C07315=1211.113,371.634,-76.951,-175.920,7.915,148.347
C07316=1211.109,371.881,-76.984,-175.919,7.917,148.348
C07317=1211.105,372.129,-77.018,-175.918,7.920,148.348
C07318=1211.101,372.377,-77.052,-175.917,7.923,148.349
C07319=1211.097,372.625,-77.085,-175.915,7.926,148.349
C07320=1211.093,372.872,-77.119,-175.914,7.929,148.349
C07321=1211.089,373.120,-77.152,-175.912,7.932,148.350
C07322=1211.085,373.368,-77.185,-175.911,7.935,148.350
C07323=1211.080,373.615,-77.220,-175.910,7.938,148.351
C07324=1211.077,373.863,-77.253,-175.909,7.941,148.351
C07325=1211.073,374.111,-77.287,-175.908,7.944,148.351
C07326=1211.068,374.359,-77.321,-175.906,7.946,148.352
C07327=1211.064,374.606,-77.355,-175.905,7.949,148.352
C07328=1211.060,374.853,-77.388,-175.904,7.952,148.353
C07329=1211.057,375.102,-77.421,-175.903,7.956,148.353
C07330=1211.052,375.349,-77.456,-175.902,7.959,148.354
C07331=1211.048,375.597,-77.489,-175.900,7.962,148.354
C07332=1211.044,375.844,-77.523,-175.899,7.964,148.354
C07333=1211.040,376.093,-77.557,-175.898,7.967,148.355
C07334=1211.036,376.340,-77.591,-175.897,7.970,148.355
C07335=1211.032,376.588,-77.624,-175.896,7.973,148.356
C07336=1211.027,376.835,-77.658,-175.894,7.976,148.356
C07337=1211.023,377.083,-77.691,-175.893,7.978,148.356
C07338=1211.020,377.331,-77.726,-175.892,7.982,148.357
C07339=1211.015,377.578,-77.760,-175.891,7.984,148.357
C07340=1211.011,377.826,-77.793,-175.890,7.987,148.358
C07341=1211.007,378.073,-77.827,-175.889,7.990,148.358
C07342=1211.003,378.322,-77.861,-175.888,7.993,148.358
C07343=1210.999,378.569,-77.895,-175.886,7.996,148.359
C07344=1210.995,378.816,-77.928,-175.886,7.999,148.359
C07345=1210.991,379.065,-77.963,-175.885,8.002,148.360
C07346=1210.987,379.312,-77.997,-175.883,8.004,148.360
C07347=1210.982,379.560,-78.031,-175.882,8.007,148.361
C07348=1210.979,379.807,-78.065,-175.881,8.010,148.361
C07349=1210.975,380.055,-78.099,-175.880,8.013,148.362
C07350=1210.971,380.303,-78.133,-175.879,8.016,148.362
C07351=1210.967,380.550,-78.167,-175.878,8.019,148.362
C07352=1210.962,380.797,-78.201,-175.877,8.022,148.363
C07353=1210.959,381.046,-78.235,-175.876,8.025,148.363
C07354=1210.955,381.293,-78.268,-175.875,8.027,148.364
C07355=1210.950,381.540,-78.303,-175.874,8.029,148.364
C07356=1210.947,381.789,-78.336,-175.873,8.033,148.365
C07357=1210.942,382.036,-78.371,-175.872,8.035,148.365
C07358=1210.938,382.283,-78.405,-175.871,8.038,148.365
C07359=1210.933,382.531,-78.438,-175.870,8.041,148.366
C07360=1210.930,382.779,-78.473,-175.869,8.044,148.366
C07361=1210.926,383.026,-78.507,-175.868,8.047,148.367
C07362=1210.922,383.274,-78.541,-175.867,8.049,148.367
C07363=1210.917,383.522,-78.575,-175.866,8.052,148.368
C07364=1210.914,383.769,-78.609,-175.866,8.055,148.368
C07365=1210.909,384.017,-78.644,-175.864,8.058,148.369
C07366=1210.906,384.265,-78.678,-175.863,8.061,148.369
C07367=1210.901,384.513,-78.711,-175.862,8.064,148.370
C07368=1210.897,384.760,-78.745,-175.862,8.066,148.370
C07369=1210.893,385.008,-78.780,-175.861,8.069,148.371
C07370=1210.889,385.255,-78.814,-175.860,8.072,148.371
C07371=1210.885,385.502,-78.849,-175.859,8.075,148.372
C07372=1210.881,385.751,-78.882,-175.858,8.078,148.372
C07373=1210.877,385.998,-78.917,-175.857,8.080,148.372
C07374=1210.873,386.245,-78.950,-175.856,8.083,148.373
C07375=1210.869,386.493,-78.985,-175.855,8.086,148.373
C07376=1210.865,386.741,-79.019,-175.854,8.089,148.374
C07377=1210.860,386.988,-79.054,-175.854,8.091,148.374
C07378=1210.857,387.236,-79.088,-175.853,8.093,148.375
C07379=1210.852,387.484,-79.122,-175.852,8.097,148.375
C07380=1210.849,387.732,-79.156,-175.851,8.099,148.376
C07381=1210.845,387.979,-79.190,-175.850,8.102,148.376
C07382=1210.840,388.227,-79.225,-175.849,8.104,148.377
C07383=1210.837,388.474,-79.259,-175.848,8.108,148.377
C07384=1210.832,388.722,-79.293,-175.848,8.110,148.378
C07385=1210.828,388.969,-79.327,-175.847,8.113,148.378
C07386=1210.824,389.217,-79.362,-175.846,8.115,148.379
C07387=1210.821,389.464,-79.396,-175.846,8.118,148.379
C07388=1210.817,389.712,-79.431,-175.844,8.121,148.380
C07389=1210.812,389.960,-79.465,-175.844,8.124,148.380
C07390=1210.808,390.207,-79.499,-175.843,8.126,148.381
C07391=1210.804,390.455,-79.534,-175.842,8.129,148.381
C07392=1210.800,390.702,-79.568,-175.842,8.131,148.382
C07393=1210.796,390.950,-79.603,-175.841,8.134,148.382
C07394=1210.792,391.197,-79.637,-175.840,8.137,148.383
C07395=1210.788,391.445,-79.671,-175.839,8.139,148.383
C07396=1210.784,391.693,-79.706,-175.839,8.142,148.384
C07397=1210.779,391.940,-79.740,-175.838,8.144,148.384
C07398=1210.776,392.188,-79.775,-175.837,8.147,148.384
C07399=1210.771,392.470,-79.813,-175.837,8.150,148.385
C07400=1210.767,392.753,-79.853,-175.836,8.153,148.386
C07401=1210.762,393.035,-79.892,-175.835,8.156,148.386
C07402=1210.757,393.317,-79.932,-175.834,8.158,148.387
C07403=1210.753,393.564,-79.966,-175.834,8.161,148.387
C07404=1210.749,393.812,-80.000,-175.832,8.164,148.388
C07405=1210.745,394.060,-80.035,-175.832,8.167,148.388
C07406=1210.742,394.308,-80.069,-175.831,8.170,148.389
C07407=1210.737,394.555,-80.104,-175.831,8.172,148.389
C07408=1210.733,394.803,-80.138,-175.830,8.175,148.390
C07409=1210.729,395.050,-80.172,-175.829,8.177,148.390
C07410=1210.725,395.298,-80.207,-175.829,8.179,148.391
C07411=1210.721,395.546,-80.242,-175.828,8.182,148.391
C07412=1210.717,395.793,-80.277,-175.828,8.184,148.391
C07413=1210.713,396.040,-80.311,-175.827,8.187,148.392
C07414=1210.709,396.288,-80.345,-175.826,8.189,148.392
C07415=1210.705,396.536,-80.380,-175.826,8.192,148.393
C07416=1210.701,396.783,-80.414,-175.825,8.195,148.394
C07417=1210.697,397.031,-80.449,-175.824,8.197,148.394
C07418=1210.692,397.279,-80.483,-175.824,8.200,148.394
C07419=1210.688,397.525,-80.519,-175.824,8.202,148.395
C07420=1210.685,397.773,-80.553,-175.823,8.205,148.395
C07421=1210.680,398.021,-80.587,-175.822,8.207,148.396
C07422=1210.676,398.269,-80.622,-175.822,8.210,148.397
C07423=1210.672,398.516,-80.657,-175.821,8.212,148.397
C07424=1210.669,398.764,-80.691,-175.821,8.214,148.397
C07425=1210.664,399.011,-80.726,-175.820,8.217,148.398
C07426=1210.660,399.259,-80.761,-175.819,8.219,148.398
C07427=1210.656,399.506,-80.795,-175.819,8.222,148.399
C07428=1210.653,399.754,-80.830,-175.818,8.224,148.399
C07429=1210.648,400.001,-80.865,-175.818,8.227,148.400
C07430=1210.644,400.249,-80.900,-175.818,8.229,148.400
C07431=1210.640,400.496,-80.934,-175.816,8.232,148.401
C07432=1210.636,400.744,-80.968,-175.816,8.234,148.401
C07433=1210.632,400.992,-81.003,-175.816,8.236,148.402
C07434=1210.628,401.239,-81.038,-175.815,8.239,148.402
C07435=1210.624,401.487,-81.073,-175.815,8.241,148.403
C07436=1210.620,401.735,-81.108,-175.814,8.244,148.403
C07437=1210.616,401.981,-81.142,-175.814,8.246,148.404
C07438=1210.612,402.229,-81.177,-175.813,8.249,148.404
C07439=1210.608,402.477,-81.212,-175.813,8.251,148.405
C07440=1210.604,402.725,-81.246,-175.812,8.253,148.405
C07441=1210.599,402.972,-81.282,-175.812,8.255,148.406
C07442=1210.595,403.220,-81.316,-175.811,8.258,148.406
C07443=1210.592,403.467,-81.350,-175.810,8.260,148.407
C07444=1210.588,403.714,-81.386,-175.810,8.263,148.407
C07445=1210.583,403.962,-81.420,-175.810,8.265,148.408
C07446=1210.579,404.210,-81.455,-175.809,8.268,148.408
C07447=1210.575,404.457,-81.490,-175.809,8.270,148.409
C07448=1210.571,404.705,-81.525,-175.808,8.272,148.409
C07449=1210.568,404.953,-81.559,-175.808,8.274,148.409
C07450=1210.564,405.200,-81.595,-175.807,8.277,148.410
C07451=1210.560,405.448,-81.629,-175.807,8.280,148.411
C07452=1210.555,405.695,-81.664,-175.806,8.282,148.411
C07453=1210.551,405.943,-81.699,-175.806,8.284,148.411
C07454=1210.547,406.190,-81.734,-175.806,8.286,148.412
C07455=1210.544,406.438,-81.768,-175.805,8.288,148.412
C07456=1210.539,406.685,-81.803,-175.805,8.290,148.413
C07457=1210.535,406.933,-81.838,-175.804,8.293,148.413
C07458=1210.531,407.179,-81.873,-175.803,8.295,148.414
C07459=1210.527,407.428,-81.908,-175.803,8.298,148.414
C07460=1210.523,407.676,-81.943,-175.803,8.300,148.415
C07461=1210.519,407.923,-81.978,-175.802,8.302,148.415
C07462=1210.515,408.171,-82.013,-175.802,8.304,148.416
C07463=1210.511,408.417,-82.048,-175.802,8.306,148.416
C07464=1210.508,408.665,-82.082,-175.801,8.309,148.417
C07465=1210.503,408.912,-82.118,-175.800,8.312,148.417
C07466=1210.499,409.160,-82.152,-175.800,8.314,148.417
C07467=1210.495,409.408,-82.187,-175.800,8.316,148.418
C07468=1210.491,409.655,-82.222,-175.799,8.318,148.419
C07469=1210.487,409.903,-82.257,-175.799,8.320,148.419
C07470=1210.483,410.150,-82.292,-175.798,8.322,148.419
C07471=1210.479,410.398,-82.327,-175.798,8.325,148.420
C07472=1210.475,410.645,-82.362,-175.798,8.327,148.420
C07473=1210.471,410.893,-82.397,-175.797,8.329,148.421
C07474=1210.467,411.141,-82.433,-175.797,8.331,148.421
C07475=1210.463,411.388,-82.467,-175.797,8.333,148.422
C07476=1210.459,411.635,-82.502,-175.796,8.335,148.422
C07477=1210.455,411.883,-82.537,-175.796,8.338,148.423
C07478=1210.451,412.130,-82.572,-175.795,8.340,148.423
C07479=1210.447,412.378,-82.607,-175.795,8.343,148.424
C07480=1210.443,412.625,-82.642,-175.794,8.345,148.424
C07481=1210.439,412.873,-82.677,-175.794,8.347,148.425
C07482=1210.435,413.120,-82.712,-175.794,8.349,148.425
C07483=1210.431,413.368,-82.747,-175.793,8.351,148.425
C07484=1210.427,413.616,-82.783,-175.793,8.353,148.426
C07485=1210.423,413.863,-82.817,-175.793,8.356,148.426
C07486=1210.419,414.110,-82.853,-175.792,8.358,148.427
C07487=1210.414,414.358,-82.887,-175.792,8.360,148.427
C07488=1210.411,414.605,-82.923,-175.791,8.362,148.428
C07489=1210.407,414.853,-82.958,-175.791,8.364,148.428
C07490=1210.402,415.100,-82.993,-175.791,8.366,148.429
C07491=1210.399,415.348,-83.028,-175.790,8.368,148.429
C07492=1210.394,415.595,-83.063,-175.790,8.371,148.430
C07493=1210.391,415.843,-83.098,-175.789,8.373,148.430
C07494=1210.387,416.091,-83.133,-175.789,8.375,148.430
C07495=1210.383,416.341,-83.169,-175.789,8.377,148.431
C07496=1210.379,416.592,-83.204,-175.788,8.379,148.431
C07497=1210.377,416.842,-83.239,-175.788,8.381,148.432
C07498=1210.379,417.093,-83.274,-175.788,8.383,148.432
C07499=1209.957,417.093,-83.312,-175.791,8.393,148.436
C07500=1209.956,416.839,-83.276,-175.791,8.392,148.436
C07501=1209.957,416.587,-83.240,-175.791,8.390,148.435
C07502=1209.961,416.333,-83.204,-175.791,8.388,148.435
C07503=1209.965,416.080,-83.168,-175.792,8.386,148.434
C07504=1209.969,415.832,-83.133,-175.792,8.383,148.434
C07505=1209.973,415.585,-83.098,-175.793,8.381,148.433
C07506=1209.977,415.337,-83.063,-175.793,8.379,148.433
C07507=1209.981,415.090,-83.028,-175.793,8.377,148.432
C07508=1209.985,414.842,-82.993,-175.794,8.375,148.432
C07509=1209.989,414.594,-82.957,-175.794,8.373,148.431
C07510=1209.993,414.347,-82.922,-175.794,8.370,148.431
C07511=1209.997,414.099,-82.887,-175.795,8.368,148.431
C07512=1210.001,413.853,-82.852,-175.795,8.366,148.430
C07513=1210.005,413.604,-82.817,-175.796,8.364,148.430
C07514=1210.009,413.357,-82.782,-175.796,8.362,148.429
C07515=1210.013,413.109,-82.747,-175.796,8.360,148.429
C07516=1210.017,412.862,-82.712,-175.797,8.358,148.428
C07517=1210.022,412.615,-82.677,-175.797,8.355,148.428
C07518=1210.025,412.367,-82.642,-175.798,8.353,148.427
C07519=1210.029,412.119,-82.607,-175.798,8.351,148.427
C07520=1210.034,411.872,-82.572,-175.798,8.349,148.426
C07521=1210.038,411.624,-82.537,-175.799,8.347,148.426
C07522=1210.042,411.377,-82.502,-175.800,8.344,148.425
C07523=1210.045,411.129,-82.467,-175.800,8.341,148.425
C07524=1210.049,410.882,-82.432,-175.801,8.339,148.425
C07525=1210.053,410.635,-82.397,-175.801,8.337,148.424
C07526=1210.057,410.387,-82.362,-175.801,8.335,148.423
C07527=1210.061,410.140,-82.327,-175.802,8.333,148.423
C07528=1210.065,409.892,-82.292,-175.802,8.331,148.423
C07529=1210.070,409.645,-82.257,-175.802,8.328,148.422
C07530=1210.073,409.397,-82.222,-175.803,8.326,148.422
C07531=1210.077,409.149,-82.187,-175.803,8.324,148.421
C07532=1210.082,408.902,-82.152,-175.803,8.322,148.421
C07533=1210.086,408.654,-82.117,-175.804,8.320,148.420
C07534=1210.090,408.407,-82.082,-175.804,8.318,148.420
C07535=1210.093,408.160,-82.048,-175.805,8.315,148.419
C07536=1210.098,407.912,-82.013,-175.806,8.313,148.419
C07537=1210.101,407.665,-81.978,-175.806,8.310,148.418
C07538=1210.105,407.416,-81.943,-175.806,8.308,148.418
C07539=1210.110,407.170,-81.908,-175.807,8.306,148.417
C07540=1210.114,406.922,-81.873,-175.807,8.304,148.417
C07541=1210.118,406.675,-81.838,-175.807,8.302,148.416
C07542=1210.122,406.427,-81.803,-175.808,8.299,148.416
C07543=1210.126,406.180,-81.769,-175.809,8.296,148.415
C07544=1210.129,405.932,-81.733,-175.809,8.294,148.415
C07545=1210.134,405.685,-81.699,-175.809,8.292,148.415
C07546=1210.138,405.436,-81.664,-175.810,8.290,148.414
C07547=1210.141,405.189,-81.628,-175.810,8.288,148.414
C07548=1210.146,404.942,-81.594,-175.811,8.285,148.413
C07549=1210.150,404.694,-81.558,-175.811,8.283,148.413
C07550=1210.154,404.447,-81.525,-175.811,8.280,148.412
C07551=1210.157,404.199,-81.490,-175.812,8.278,148.412
C07552=1210.162,403.952,-81.455,-175.812,8.276,148.411
C07553=1210.166,403.704,-81.420,-175.813,8.273,148.411
C07554=1210.170,403.456,-81.385,-175.814,8.271,148.410
C07555=1210.174,403.209,-81.350,-175.814,8.269,148.410
C07556=1210.178,402.962,-81.316,-175.814,8.266,148.409
C07557=1210.182,402.714,-81.281,-175.815,8.264,148.409
C07558=1210.186,402.466,-81.247,-175.816,8.261,148.408
C07559=1210.190,402.219,-81.211,-175.816,8.259,148.408
C07560=1210.195,401.971,-81.177,-175.816,8.257,148.407
C07561=1210.199,401.723,-81.142,-175.817,8.254,148.407
C07562=1210.202,401.477,-81.107,-175.817,8.252,148.406
C07563=1210.206,401.229,-81.072,-175.818,8.250,148.406
C07564=1210.211,400.981,-81.038,-175.819,8.247,148.405
C07565=1210.215,400.733,-81.003,-175.819,8.244,148.405
C07566=1210.219,400.486,-80.968,-175.820,8.242,148.404
C07567=1210.222,400.239,-80.934,-175.820,8.240,148.404
C07568=1210.227,399.991,-80.899,-175.821,8.237,148.403
C07569=1210.231,399.743,-80.864,-175.821,8.235,148.403
C07570=1210.235,399.496,-80.829,-175.822,8.233,148.402
C07571=1210.238,399.248,-80.795,-175.822,8.230,148.402
C07572=1210.243,399.001,-80.760,-175.823,8.228,148.402
C07573=1210.247,398.753,-80.726,-175.824,8.225,148.401
C07574=1210.251,398.505,-80.691,-175.824,8.222,148.400
C07575=1210.254,398.258,-80.656,-175.825,8.220,148.400
C07576=1210.259,398.011,-80.622,-175.825,8.217,148.399
C07577=1210.263,397.763,-80.587,-175.826,8.215,148.399
C07578=1210.267,397.515,-80.552,-175.826,8.213,148.399
C07579=1210.270,397.267,-80.518,-175.827,8.210,148.398
C07580=1210.275,397.021,-80.483,-175.827,8.208,148.397
C07581=1210.279,396.773,-80.448,-175.828,8.205,148.397
C07582=1210.283,396.525,-80.414,-175.829,8.203,148.397
C07583=1210.286,396.277,-80.379,-175.829,8.199,148.396
C07584=1210.291,396.030,-80.345,-175.830,8.198,148.396
C07585=1210.295,395.782,-80.310,-175.830,8.195,148.395
C07586=1210.300,395.534,-80.276,-175.831,8.192,148.395
C07587=1210.303,395.287,-80.242,-175.832,8.190,148.394
C07588=1210.307,395.040,-80.206,-175.832,8.187,148.394
C07589=1210.312,394.792,-80.172,-175.833,8.185,148.393
C07590=1210.315,394.545,-80.138,-175.834,8.182,148.393
C07591=1210.319,394.297,-80.103,-175.834,8.180,148.392
C07592=1210.323,394.049,-80.068,-175.835,8.177,148.392
C07593=1210.327,393.802,-80.034,-175.835,8.175,148.391
C07594=1210.331,393.554,-80.000,-175.837,8.172,148.391
C07595=1210.336,393.306,-79.965,-175.837,8.170,148.390
C07596=1210.340,393.024,-79.925,-175.838,8.166,148.390
C07597=1210.345,392.742,-79.887,-175.838,8.163,148.389
C07598=1210.349,392.460,-79.847,-175.839,8.161,148.389
C07599=1210.354,392.177,-79.809,-175.840,8.157,148.388
C07600=1210.358,391.929,-79.774,-175.840,8.155,148.387
C07601=1210.363,391.682,-79.739,-175.842,8.152,148.387
C07602=1210.366,391.434,-79.705,-175.842,8.149,148.386
C07603=1210.370,391.187,-79.671,-175.843,8.147,148.386
C07604=1210.374,390.940,-79.637,-175.844,8.144,148.386
C07605=1210.378,390.691,-79.602,-175.844,8.142,148.385
C07606=1210.383,390.444,-79.567,-175.845,8.139,148.385
C07607=1210.386,390.196,-79.533,-175.846,8.136,148.384
C07608=1210.390,389.949,-79.499,-175.847,8.134,148.384
C07609=1210.395,389.701,-79.464,-175.847,8.131,148.383
C07610=1210.398,389.454,-79.430,-175.849,8.128,148.383
C07611=1210.403,389.206,-79.396,-175.849,8.126,148.382
C07612=1210.406,388.958,-79.361,-175.850,8.123,148.382
C07613=1210.411,388.711,-79.327,-175.851,8.120,148.381
C07614=1210.415,388.464,-79.293,-175.851,8.118,148.381
C07615=1210.418,388.216,-79.258,-175.852,8.115,148.380
C07616=1210.423,387.968,-79.224,-175.853,8.112,148.380
C07617=1210.427,387.721,-79.190,-175.854,8.110,148.379
C07618=1210.431,387.473,-79.155,-175.855,8.107,148.379
C07619=1210.435,387.226,-79.121,-175.856,8.104,148.378
C07620=1210.439,386.977,-79.087,-175.856,8.102,148.378
C07621=1210.443,386.730,-79.053,-175.857,8.099,148.377
C07622=1210.447,386.483,-79.019,-175.858,8.096,148.377
C07623=1210.451,386.235,-78.984,-175.859,8.093,148.376
C07624=1210.455,385.987,-78.950,-175.860,8.091,148.376
C07625=1210.460,385.740,-78.915,-175.860,8.088,148.375
C07626=1210.463,385.492,-78.881,-175.861,8.085,148.375
C07627=1210.468,385.244,-78.847,-175.862,8.082,148.374
C07628=1210.472,384.997,-78.814,-175.863,8.079,148.374
C07629=1210.476,384.749,-78.779,-175.864,8.077,148.374
C07630=1210.479,384.502,-78.745,-175.865,8.074,148.373
C07631=1210.484,384.254,-78.710,-175.866,8.071,148.373
C07632=1210.488,384.006,-78.677,-175.867,8.068,148.372
C07633=1210.492,383.759,-78.642,-175.868,8.065,148.372
C07634=1210.496,383.511,-78.609,-175.869,8.062,148.371
C07635=1210.500,383.263,-78.574,-175.869,8.060,148.371
C07636=1210.504,383.016,-78.540,-175.871,8.057,148.370
C07637=1210.509,382.768,-78.506,-175.872,8.054,148.370
C07638=1210.512,382.520,-78.472,-175.873,8.051,148.369
C07639=1210.516,382.273,-78.438,-175.874,8.049,148.369
C07640=1210.521,382.025,-78.404,-175.875,8.046,148.369
C07641=1210.524,381.777,-78.370,-175.876,8.043,148.368
C07642=1210.528,381.530,-78.336,-175.876,8.041,148.368
C07643=1210.532,381.283,-78.302,-175.878,8.038,148.367
C07644=1210.537,381.035,-78.268,-175.878,8.035,148.367
C07645=1210.540,380.787,-78.234,-175.880,8.032,148.366
C07646=1210.545,380.540,-78.199,-175.881,8.029,148.366
C07647=1210.549,380.292,-78.166,-175.881,8.026,148.365
C07648=1210.552,380.044,-78.132,-175.883,8.023,148.365
C07649=1210.557,379.797,-78.097,-175.884,8.020,148.365
C07650=1210.561,379.549,-78.064,-175.885,8.018,148.364
C07651=1210.566,379.301,-78.030,-175.886,8.014,148.364
C07652=1210.569,379.053,-77.996,-175.887,8.012,148.363
C07653=1210.573,378.806,-77.962,-175.888,8.009,148.363
C07654=1210.577,378.559,-77.928,-175.889,8.006,148.362
C07655=1210.582,378.311,-77.895,-175.891,8.003,148.362
C07656=1210.586,378.063,-77.860,-175.891,8.000,148.361
C07657=1210.590,377.815,-77.827,-175.893,7.997,148.361
C07658=1210.594,377.568,-77.793,-175.894,7.994,148.361
C07659=1210.598,377.320,-77.758,-175.895,7.992,148.360
C07660=1210.602,377.072,-77.725,-175.896,7.989,148.360
C07661=1210.605,376.825,-77.691,-175.897,7.986,148.359
C07662=1210.610,376.577,-77.657,-175.898,7.983,148.359
C07663=1210.614,376.330,-77.623,-175.899,7.980,148.358
C07664=1210.618,376.081,-77.590,-175.901,7.977,148.358
C07665=1210.622,375.834,-77.555,-175.902,7.974,148.358
C07666=1210.626,375.586,-77.522,-175.903,7.972,148.357
C07667=1210.630,375.339,-77.488,-175.904,7.969,148.357
C07668=1210.635,375.090,-77.454,-175.905,7.966,148.357
C07669=1210.638,374.843,-77.420,-175.907,7.962,148.356
C07670=1210.643,374.595,-77.387,-175.908,7.960,148.356
C07671=1210.646,374.348,-77.353,-175.909,7.957,148.355
C07672=1210.651,374.100,-77.320,-175.910,7.954,148.355
C07673=1210.654,373.853,-77.285,-175.911,7.951,148.354
C07674=1210.659,373.605,-77.252,-175.913,7.948,148.354
C07675=1210.663,373.357,-77.218,-175.914,7.945,148.354
C07676=1210.667,373.110,-77.185,-175.915,7.942,148.353
C07677=1210.671,372.862,-77.151,-175.917,7.939,148.353
C07678=1210.675,372.614,-77.117,-175.918,7.936,148.352
C07679=1210.679,372.366,-77.084,-175.919,7.933,148.352
C07680=1210.684,372.118,-77.050,-175.920,7.930,148.352
C07681=1210.688,371.871,-77.016,-175.922,7.928,148.351
C07682=1210.692,371.623,-76.983,-175.923,7.925,148.351
C07683=1210.696,371.376,-76.950,-175.925,7.921,148.350
C07684=1210.700,371.128,-76.915,-175.926,7.919,148.350
C07685=1210.704,370.880,-76.882,-175.927,7.916,148.350
C07686=1210.708,370.632,-76.849,-175.929,7.913,148.349
C07687=1210.712,370.385,-76.815,-175.930,7.910,148.349
C07688=1210.716,370.137,-76.782,-175.932,7.906,148.348
C07689=1210.721,369.889,-76.748,-175.933,7.904,148.348
C07690=1210.724,369.641,-76.714,-175.934,7.901,148.348
C07691=1210.728,369.394,-76.681,-175.936,7.898,148.348
C07692=1210.732,369.146,-76.648,-175.937,7.895,148.347
C07693=1210.737,368.898,-76.614,-175.939,7.892,148.347
C07694=1210.740,368.651,-76.581,-175.940,7.889,148.346
C07695=1210.745,368.403,-76.547,-175.941,7.886,148.346
C07696=1210.749,368.155,-76.514,-175.943,7.883,148.345
C07697=1210.754,367.908,-76.481,-175.944,7.880,148.345
C07698=1210.757,367.659,-76.447,-175.946,7.877,148.345
C07699=1210.761,367.412,-76.413,-175.947,7.874,148.344
C07700=1210.766,367.132,-76.376,-175.948,7.871,148.344
C07701=1210.771,366.851,-76.338,-175.950,7.867,148.344
C07702=1210.775,366.572,-76.300,-175.952,7.864,148.343
C07703=1210.779,366.291,-76.263,-175.954,7.861,148.343
C07704=1210.784,366.043,-76.229,-175.955,7.857,148.343
C07705=1210.788,365.796,-76.195,-175.957,7.855,148.342
C07706=1210.792,365.548,-76.162,-175.958,7.852,148.342
C07707=1210.796,365.300,-76.129,-175.960,7.848,148.341
C07708=1210.801,365.052,-76.096,-175.961,7.846,148.341
C07709=1210.805,364.805,-76.063,-175.963,7.843,148.341
C07710=1210.809,364.557,-76.030,-175.965,7.839,148.340
C07711=1210.813,364.309,-75.997,-175.966,7.837,148.340
C07712=1210.817,364.061,-75.963,-175.967,7.834,148.340
C07713=1210.821,363.813,-75.930,-175.969,7.830,148.339
C07714=1210.825,363.565,-75.897,-175.971,7.828,148.339
C07715=1210.829,363.318,-75.864,-175.972,7.825,148.339
C07716=1210.833,363.070,-75.830,-175.974,7.821,148.338
C07717=1210.837,362.822,-75.797,-175.975,7.819,148.338
C07718=1210.841,362.574,-75.764,-175.977,7.815,148.338
C07719=1210.845,362.327,-75.731,-175.979,7.813,148.338
C07720=1210.850,362.079,-75.698,-175.980,7.810,148.337
C07721=1210.854,361.831,-75.665,-175.982,7.807,148.337
C07722=1210.858,361.584,-75.631,-175.983,7.804,148.337
C07723=1210.862,361.336,-75.598,-175.985,7.801,148.336
C07724=1210.866,361.088,-75.565,-175.987,7.798,148.336
C07725=1210.870,360.840,-75.532,-175.988,7.795,148.336
C07726=1210.874,360.593,-75.499,-175.990,7.791,148.335
C07727=1210.878,360.345,-75.466,-175.992,7.789,148.335
C07728=1210.882,360.098,-75.433,-175.994,7.785,148.335
C07729=1210.886,359.850,-75.400,-175.995,7.783,148.335
C07730=1210.891,359.601,-75.368,-175.996,7.780,148.334
C07731=1210.895,359.354,-75.334,-175.999,7.777,148.334
C07732=1210.899,359.106,-75.301,-176.000,7.774,148.334
C07733=1210.903,358.858,-75.268,-176.002,7.770,148.333
C07734=1210.907,358.611,-75.235,-176.004,7.768,148.333
C07735=1210.911,358.363,-75.202,-176.005,7.764,148.333
C07736=1210.915,358.115,-75.170,-176.007,7.762,148.333
C07737=1210.919,357.867,-75.137,-176.008,7.759,148.332
C07738=1210.923,357.619,-75.104,-176.011,7.756,148.332
C07739=1210.927,357.372,-75.070,-176.012,7.753,148.332
C07740=1210.932,357.123,-75.038,-176.014,7.749,148.331
C07741=1210.936,356.875,-75.005,-176.016,7.747,148.331
C07742=1210.940,356.628,-74.972,-176.018,7.744,148.331
C07743=1210.943,356.380,-74.939,-176.019,7.741,148.330
C07744=1210.949,356.133,-74.907,-176.021,7.737,148.330
C07745=1210.953,355.885,-74.874,-176.023,7.735,148.330
C07746=1210.957,355.637,-74.841,-176.025,7.732,148.330
C07747=1210.961,355.389,-74.808,-176.026,7.729,148.329
C07748=1210.965,355.141,-74.776,-176.028,7.726,148.329
C07749=1210.969,354.894,-74.743,-176.030,7.723,148.329
C07750=1210.973,354.645,-74.710,-176.031,7.720,148.329
C07751=1210.977,354.398,-74.677,-176.034,7.717,148.328
C07752=1210.981,354.150,-74.644,-176.035,7.714,148.328
C07753=1210.985,353.902,-74.612,-176.037,7.711,148.328
C07754=1210.989,353.654,-74.579,-176.039,7.708,148.328
C07755=1210.994,353.407,-74.547,-176.041,7.705,148.327
C07756=1210.998,353.159,-74.514,-176.042,7.702,148.327
C07757=1211.002,352.911,-74.481,-176.045,7.699,148.327
C07758=1211.006,352.663,-74.449,-176.046,7.696,148.327
C07759=1211.011,352.415,-74.415,-176.048,7.693,148.327
C07760=1211.014,352.167,-74.384,-176.050,7.690,148.326
C07761=1211.018,351.920,-74.350,-176.052,7.687,148.326
C07762=1211.023,351.671,-74.318,-176.054,7.684,148.326
C07763=1211.027,351.424,-74.286,-176.056,7.681,148.326
C07764=1211.031,351.176,-74.253,-176.057,7.678,148.325
C07765=1211.035,350.928,-74.220,-176.060,7.675,148.325
C07766=1211.039,350.680,-74.188,-176.061,7.672,148.325
C07767=1211.043,350.433,-74.155,-176.063,7.669,148.325
C07768=1211.048,350.184,-74.123,-176.065,7.666,148.324
C07769=1211.052,349.938,-74.091,-176.067,7.663,148.324
C07770=1211.056,349.689,-74.058,-176.068,7.660,148.324
C07771=1211.061,349.441,-74.026,-176.071,7.657,148.324
C07772=1211.064,349.193,-73.993,-176.072,7.655,148.324
C07773=1211.068,348.945,-73.961,-176.075,7.651,148.323
C07774=1211.073,348.698,-73.928,-176.076,7.649,148.323
C07775=1211.077,348.450,-73.896,-176.078,7.645,148.323
C07776=1211.081,348.202,-73.864,-176.080,7.643,148.323
C07777=1211.085,347.954,-73.831,-176.082,7.640,148.322
C07778=1211.089,347.706,-73.799,-176.084,7.637,148.322
C07779=1211.093,347.459,-73.767,-176.086,7.634,148.322
C07780=1211.098,347.211,-73.734,-176.088,7.631,148.322
C07781=1211.102,346.962,-73.702,-176.090,7.628,148.322
C07782=1211.106,346.714,-73.670,-176.092,7.625,148.321
C07783=1211.110,346.466,-73.637,-176.094,7.622,148.321
C07784=1211.114,346.219,-73.605,-176.095,7.619,148.321
C07785=1211.119,345.971,-73.573,-176.098,7.616,148.321
C07786=1211.122,345.723,-73.541,-176.099,7.614,148.321
C07787=1211.127,345.475,-73.508,-176.102,7.610,148.320
C07788=1211.131,345.228,-73.476,-176.103,7.608,148.320
C07789=1211.135,344.980,-73.444,-176.105,7.604,148.320
C07790=1211.139,344.732,-73.412,-176.107,7.602,148.320
C07791=1211.144,344.484,-73.380,-176.109,7.599,148.320
C07792=1211.148,344.236,-73.348,-176.111,7.596,148.319
C07793=1211.152,343.988,-73.315,-176.113,7.593,148.319
C07794=1211.156,343.740,-73.283,-176.115,7.590,148.319
C07795=1211.161,343.492,-73.251,-176.117,7.587,148.319
C07796=1211.164,343.244,-73.219,-176.120,7.584,148.319
C07797=1211.169,342.996,-73.187,-176.121,7.581,148.319
C07798=1211.173,342.749,-73.155,-176.124,7.578,148.318
C07799=1211.177,342.500,-73.123,-176.125,7.575,148.318
C07800=1211.181,342.252,-73.091,-176.127,7.572,148.318
C07801=1211.185,342.004,-73.059,-176.129,7.570,148.318
C07802=1211.190,341.757,-73.026,-176.131,7.566,148.318
C07803=1211.193,341.509,-72.994,-176.133,7.564,148.318
C07804=1211.199,341.231,-72.959,-176.136,7.561,148.317
C07805=1211.203,340.953,-72.923,-176.138,7.557,148.317
C07806=1211.207,340.675,-72.887,-176.140,7.554,148.317
C07807=1211.213,340.396,-72.851,-176.142,7.551,148.317
C07808=1211.217,340.148,-72.819,-176.145,7.548,148.317
C07809=1211.221,339.901,-72.788,-176.146,7.545,148.317
C07810=1211.225,339.652,-72.755,-176.149,7.542,148.316
C07811=1211.229,339.404,-72.724,-176.150,7.539,148.316
C07812=1211.233,339.157,-72.692,-176.153,7.536,148.316
C07813=1211.238,338.909,-72.660,-176.155,7.534,148.316
C07814=1211.242,338.661,-72.628,-176.157,7.530,148.316
C07815=1211.246,338.413,-72.596,-176.159,7.528,148.316
C07816=1211.250,338.165,-72.564,-176.161,7.524,148.315
C07817=1211.255,337.918,-72.532,-176.163,7.522,148.315
C07818=1211.258,337.670,-72.501,-176.165,7.519,148.315
C07819=1211.262,337.422,-72.469,-176.167,7.515,148.315
C07820=1211.267,337.173,-72.437,-176.169,7.513,148.315
C07821=1211.271,336.925,-72.406,-176.172,7.510,148.315
C07822=1211.275,336.678,-72.374,-176.173,7.507,148.315
C07823=1211.279,336.430,-72.342,-176.175,7.504,148.314
C07824=1211.283,336.182,-72.310,-176.178,7.502,148.314
C07825=1211.288,335.934,-72.279,-176.180,7.498,148.314
C07826=1211.292,335.686,-72.247,-176.181,7.496,148.314
C07827=1211.296,335.438,-72.216,-176.184,7.493,148.314
C07828=1211.301,335.190,-72.183,-176.186,7.490,148.314
C07829=1211.305,334.943,-72.152,-176.188,7.487,148.314
C07830=1211.309,334.694,-72.121,-176.191,7.484,148.314
C07831=1211.313,334.446,-72.089,-176.192,7.481,148.313
C07832=1211.317,334.198,-72.057,-176.194,7.478,148.313
C07833=1211.321,333.950,-72.026,-176.197,7.476,148.313
C07834=1211.326,333.702,-71.994,-176.199,7.473,148.313
C07835=1211.330,333.454,-71.962,-176.201,7.470,148.313
C07836=1211.334,333.206,-71.931,-176.203,7.467,148.313
C07837=1211.338,332.958,-71.900,-176.205,7.465,148.313
C07838=1211.342,332.711,-71.868,-176.207,7.461,148.313
C07839=1211.346,332.462,-71.837,-176.210,7.458,148.312
C07840=1211.351,332.215,-71.806,-176.212,7.456,148.312
C07841=1211.355,331.966,-71.773,-176.214,7.453,148.312
C07842=1211.360,331.719,-71.742,-176.216,7.450,148.312
C07843=1211.363,331.470,-71.710,-176.218,7.447,148.312
C07844=1211.368,331.223,-71.680,-176.220,7.444,148.312
C07845=1211.372,330.974,-71.648,-176.223,7.441,148.312
C07846=1211.376,330.727,-71.617,-176.224,7.439,148.312
C07847=1211.380,330.478,-71.585,-176.227,7.436,148.312
C07848=1211.385,330.231,-71.555,-176.229,7.433,148.312
C07849=1211.388,329.982,-71.523,-176.231,7.430,148.312
C07850=1211.393,329.735,-71.492,-176.233,7.427,148.311
C07851=1211.397,329.486,-71.460,-176.236,7.425,148.311
C07852=1211.401,329.239,-71.429,-176.238,7.421,148.311
C07853=1211.405,328.990,-71.397,-176.240,7.419,148.311
C07854=1211.410,328.743,-71.367,-176.242,7.416,148.311
C07855=1211.413,328.494,-71.335,-176.244,7.414,148.311
C07856=1211.418,328.247,-71.304,-176.246,7.410,148.311
C07857=1211.422,327.998,-71.272,-176.248,7.408,148.311
C07858=1211.426,327.751,-71.241,-176.251,7.405,148.311
C07859=1211.431,327.503,-71.211,-176.253,7.402,148.311
C07860=1211.435,327.255,-71.179,-176.255,7.399,148.310
C07861=1211.439,327.007,-71.148,-176.258,7.396,148.310
C07862=1211.443,326.759,-71.116,-176.259,7.394,148.310
C07863=1211.447,326.511,-71.085,-176.262,7.391,148.310
C07864=1211.451,326.262,-71.054,-176.264,7.388,148.310
C07865=1211.456,326.015,-71.023,-176.266,7.385,148.310
C07866=1211.460,325.767,-70.992,-176.268,7.383,148.310
C07867=1211.464,325.518,-70.961,-176.271,7.379,148.310
C07868=1211.469,325.270,-70.930,-176.273,7.376,148.310
C07869=1211.473,325.022,-70.898,-176.275,7.374,148.310
C07870=1211.477,324.774,-70.868,-176.278,7.371,148.310
C07871=1211.481,324.526,-70.837,-176.279,7.368,148.310
C07872=1211.485,324.278,-70.806,-176.282,7.365,148.310
C07873=1211.490,324.030,-70.775,-176.284,7.363,148.310
C07874=1211.494,323.782,-70.744,-176.286,7.360,148.309
C07875=1211.498,323.534,-70.713,-176.288,7.358,148.309
C07876=1211.503,323.286,-70.682,-176.291,7.355,148.309
C07877=1211.507,323.037,-70.651,-176.293,7.351,148.309
C07878=1211.510,322.790,-70.620,-176.295,7.349,148.309
C07879=1211.515,322.542,-70.589,-176.298,7.346,148.309
C07880=1211.519,322.293,-70.558,-176.300,7.343,148.309
C07881=1211.524,322.046,-70.527,-176.302,7.340,148.309
C07882=1211.528,321.798,-70.497,-176.304,7.338,148.309
C07883=1211.531,321.549,-70.466,-176.307,7.335,148.309
C07884=1211.536,321.301,-70.435,-176.309,7.333,148.309
C07885=1211.541,321.053,-70.405,-176.311,7.329,148.309
C07886=1211.544,320.805,-70.373,-176.313,7.327,148.309
C07887=1211.548,320.558,-70.343,-176.316,7.324,148.309
C07888=1211.553,320.310,-70.312,-176.318,7.321,148.309
C07889=1211.557,320.061,-70.281,-176.320,7.318,148.309
C07890=1211.562,319.813,-70.250,-176.323,7.315,148.309
C07891=1211.565,319.565,-70.220,-176.325,7.313,148.309
C07892=1211.570,319.317,-70.189,-176.327,7.310,148.309
C07893=1211.574,319.069,-70.158,-176.329,7.308,148.309
C07894=1211.579,318.821,-70.127,-176.332,7.305,148.309
C07895=1211.582,318.573,-70.097,-176.334,7.302,148.308
C07896=1211.587,318.325,-70.066,-176.336,7.299,148.308
C07897=1211.591,318.077,-70.035,-176.339,7.296,148.308
C07898=1211.595,317.828,-70.006,-176.341,7.294,148.308
C07899=1211.600,317.580,-69.975,-176.343,7.290,148.308
C07900=1211.604,317.332,-69.944,-176.345,7.288,148.308
C07901=1211.608,317.084,-69.914,-176.348,7.285,148.308
C07902=1211.612,316.836,-69.883,-176.350,7.283,148.308
C07903=1211.617,316.588,-69.852,-176.352,7.280,148.308
C07904=1211.621,316.340,-69.822,-176.355,7.277,148.308
C07905=1211.625,316.092,-69.791,-176.357,7.274,148.308
C07906=1211.629,315.844,-69.761,-176.359,7.272,148.308
C07907=1211.634,315.596,-69.731,-176.362,7.269,148.308
C07908=1211.638,315.320,-69.696,-176.364,7.266,148.308
C07909=1211.644,315.043,-69.663,-176.367,7.263,148.308
C07910=1211.648,314.768,-69.628,-176.370,7.260,148.308
C07911=1211.652,314.492,-69.595,-176.372,7.257,148.308
C07912=1211.657,314.243,-69.564,-176.374,7.255,148.308
C07913=1211.661,313.995,-69.534,-176.377,7.251,148.308
C07914=1211.665,313.747,-69.503,-176.379,7.249,148.308
C07915=1211.670,313.499,-69.473,-176.381,7.246,148.308
C07916=1211.674,313.251,-69.443,-176.383,7.244,148.308
C07917=1211.679,313.003,-69.412,-176.386,7.241,148.308
C07918=1211.682,312.755,-69.382,-176.388,7.239,148.308
C07919=1211.687,312.506,-69.352,-176.391,7.235,148.308
C07920=1211.691,312.258,-69.322,-176.394,7.232,148.308
C07921=1211.695,312.011,-69.291,-176.395,7.230,148.308
C07922=1211.699,311.762,-69.261,-176.398,7.227,148.308
C07923=1211.704,311.514,-69.231,-176.400,7.225,148.308
C07924=1211.708,311.266,-69.201,-176.403,7.222,148.308
C07925=1211.712,311.017,-69.170,-176.405,7.219,148.308
C07926=1211.716,310.770,-69.140,-176.407,7.216,148.308
C07927=1211.721,310.521,-69.110,-176.410,7.214,148.308
C07928=1211.725,310.273,-69.080,-176.412,7.211,148.308
C07929=1211.729,310.025,-69.050,-176.414,7.209,148.308
C07930=1211.734,309.777,-69.019,-176.417,7.206,148.308
C07931=1211.738,309.529,-68.990,-176.419,7.203,148.308
C07932=1211.743,309.281,-68.959,-176.421,7.200,148.308
C07933=1211.747,309.033,-68.930,-176.424,7.198,148.308
C07934=1211.750,308.784,-68.899,-176.426,7.195,148.308
C07935=1211.755,308.536,-68.869,-176.428,7.193,148.308
C07936=1211.759,308.288,-68.839,-176.431,7.190,148.308
C07937=1211.764,308.040,-68.809,-176.433,7.188,148.308
C07938=1211.768,307.792,-68.779,-176.436,7.185,148.308
C07939=1211.772,307.544,-68.749,-176.438,7.182,148.308
C07940=1211.776,307.296,-68.719,-176.441,7.179,148.308
C07941=1211.781,307.047,-68.689,-176.443,7.176,148.308
C07942=1211.785,306.799,-68.660,-176.445,7.174,148.308
C07943=1211.789,306.551,-68.629,-176.448,7.171,148.308
C07944=1211.794,306.303,-68.600,-176.450,7.169,148.308
C07945=1211.798,306.055,-68.570,-176.452,7.166,148.308
C07946=1211.802,305.807,-68.539,-176.455,7.163,148.308
C07947=1211.807,305.558,-68.510,-176.457,7.160,148.308
C07948=1211.811,305.310,-68.480,-176.459,7.158,148.308
C07949=1211.815,305.062,-68.450,-176.462,7.155,148.308
C07950=1211.819,304.814,-68.420,-176.464,7.153,148.308
C07951=1211.824,304.566,-68.391,-176.467,7.150,148.308
C07952=1211.828,304.318,-68.361,-176.469,7.148,148.308
C07953=1211.832,304.070,-68.331,-176.472,7.145,148.308
C07954=1211.837,303.821,-68.301,-176.474,7.142,148.308
C07955=1211.841,303.573,-68.272,-176.476,7.139,148.308
C07956=1211.845,303.325,-68.241,-176.479,7.137,148.309
C07957=1211.850,303.077,-68.211,-176.481,7.134,148.309
C07958=1211.854,302.828,-68.182,-176.483,7.132,148.309
C07959=1211.858,302.580,-68.152,-176.486,7.129,148.309
C07960=1211.862,302.332,-68.123,-176.488,7.127,148.309
C07961=1211.867,302.084,-68.092,-176.491,7.124,148.309
C07962=1211.871,301.836,-68.063,-176.493,7.121,148.309
C07963=1211.875,301.587,-68.033,-176.496,7.118,148.309
C07964=1211.879,301.339,-68.004,-176.498,7.116,148.309
C07965=1211.884,301.091,-67.974,-176.500,7.113,148.309
C07966=1211.888,300.843,-67.945,-176.503,7.111,148.309
C07967=1211.893,300.594,-67.915,-176.505,7.108,148.309
C07968=1211.897,300.346,-67.885,-176.508,7.106,148.309
C07969=1211.901,300.098,-67.856,-176.510,7.103,148.309
C07970=1211.905,299.850,-67.826,-176.513,7.101,148.309
C07971=1211.910,299.602,-67.797,-176.515,7.098,148.309
C07972=1211.914,299.354,-67.767,-176.517,7.096,148.309
C07973=1211.918,299.106,-67.738,-176.520,7.093,148.309
C07974=1211.922,298.858,-67.708,-176.522,7.090,148.309
C07975=1211.926,298.609,-67.679,-176.525,7.087,148.309
C07976=1211.931,298.361,-67.650,-176.527,7.085,148.310
C07977=1211.935,298.112,-67.619,-176.529,7.083,148.310
C07978=1211.940,297.864,-67.590,-176.532,7.080,148.310
C07979=1211.944,297.616,-67.561,-176.534,7.078,148.310
C07980=1211.949,297.368,-67.532,-176.537,7.075,148.310
C07981=1211.953,297.119,-67.503,-176.539,7.073,148.310
C07982=1211.957,296.871,-67.473,-176.542,7.070,148.310
C07983=1211.961,296.623,-67.444,-176.544,7.068,148.310
C07984=1211.966,296.375,-67.414,-176.547,7.065,148.310
C07985=1211.970,296.126,-67.385,-176.549,7.062,148.310
C07986=1211.974,295.878,-67.355,-176.552,7.059,148.310
C07987=1211.978,295.630,-67.326,-176.554,7.057,148.310
C07988=1211.983,295.382,-67.297,-176.556,7.054,148.310
C07989=1211.987,295.133,-67.268,-176.559,7.052,148.310
C07990=1211.992,294.885,-67.239,-176.562,7.049,148.310
C07991=1211.996,294.637,-67.209,-176.564,7.047,148.311
C07992=1212.000,294.389,-67.180,-176.566,7.044,148.311
C07993=1212.004,294.141,-67.151,-176.569,7.042,148.311
C07994=1212.009,293.892,-67.123,-176.571,7.039,148.311
C07995=1212.013,293.644,-67.093,-176.573,7.036,148.311
C07996=1212.017,293.396,-67.064,-176.576,7.035,148.311
C07997=1212.021,293.148,-67.034,-176.579,7.032,148.311
C07998=1212.026,292.899,-67.005,-176.581,7.029,148.311
C07999=1212.030,292.651,-66.976,-176.583,7.026,148.311
C08000=1212.035,292.403,-66.947,-176.586,7.024,148.311
C08001=1212.039,292.154,-66.918,-176.588,7.021,148.311
C08002=1212.043,291.906,-66.889,-176.591,7.019,148.311
C08003=1212.047,291.658,-66.860,-176.594,7.016,148.311
C08004=1212.052,291.410,-66.832,-176.596,7.014,148.312
C08005=1212.056,291.161,-66.802,-176.598,7.012,148.312
C08006=1212.060,290.913,-66.773,-176.600,7.009,148.312
C08007=1212.065,290.665,-66.744,-176.603,7.007,148.312
C08008=1212.069,290.417,-66.715,-176.606,7.004,148.312
C08009=1212.073,290.169,-66.686,-176.608,7.002,148.312
C08010=1212.077,289.920,-66.657,-176.611,6.999,148.312
C08011=1212.082,289.672,-66.628,-176.613,6.996,148.312
C08012=1212.087,289.398,-66.596,-176.616,6.994,148.312
C08013=1212.092,289.123,-66.565,-176.619,6.991,148.312
C08014=1212.096,288.850,-66.532,-176.621,6.988,148.312
C08015=1212.101,288.575,-66.501,-176.624,6.986,148.313
C08016=1212.105,288.326,-66.472,-176.626,6.983,148.313
C08017=1212.110,288.078,-66.443,-176.629,6.980,148.313
C08018=1212.114,287.829,-66.414,-176.631,6.977,148.313
C08019=1212.118,287.582,-66.385,-176.634,6.976,148.313
C08020=1212.123,287.333,-66.357,-176.636,6.973,148.313
C08021=1212.127,287.085,-66.327,-176.639,6.970,148.313
C08022=1212.132,286.837,-66.299,-176.641,6.968,148.313
C08023=1212.136,286.588,-66.271,-176.644,6.965,148.313
C08024=1212.140,286.340,-66.241,-176.646,6.963,148.314
C08025=1212.145,286.092,-66.213,-176.649,6.960,148.314
C08026=1212.148,285.844,-66.184,-176.651,6.958,148.314
C08027=1212.153,285.595,-66.155,-176.654,6.956,148.314
C08028=1212.158,285.347,-66.127,-176.656,6.953,148.314
C08029=1212.161,285.099,-66.098,-176.658,6.951,148.314
C08030=1212.167,284.851,-66.070,-176.661,6.948,148.314
C08031=1212.171,284.602,-66.041,-176.664,6.946,148.314
C08032=1212.174,284.354,-66.012,-176.666,6.944,148.314
C08033=1212.180,284.106,-65.984,-176.668,6.941,148.314
C08034=1212.184,283.857,-65.955,-176.671,6.939,148.314
C08035=1212.187,283.609,-65.926,-176.674,6.936,148.315
C08036=1212.193,283.360,-65.898,-176.676,6.934,148.315
C08037=1212.196,283.112,-65.870,-176.678,6.931,148.315
C08038=1212.201,282.864,-65.841,-176.681,6.929,148.315
C08039=1212.206,282.615,-65.812,-176.683,6.927,148.315
C08040=1212.209,282.367,-65.784,-176.686,6.924,148.315
C08041=1212.214,282.119,-65.755,-176.689,6.922,148.315
C08042=1212.218,281.870,-65.727,-176.691,6.919,148.316
C08043=1212.223,281.622,-65.699,-176.693,6.916,148.316
C08044=1212.227,281.373,-65.671,-176.696,6.914,148.316
C08045=1212.232,281.126,-65.642,-176.699,6.912,148.316
C08046=1212.236,280.877,-65.613,-176.701,6.909,148.316
C08047=1212.240,280.628,-65.585,-176.703,6.907,148.316
C08048=1212.244,280.380,-65.557,-176.706,6.904,148.316
C08049=1212.249,280.132,-65.528,-176.708,6.902,148.316
C08050=1212.253,279.884,-65.500,-176.710,6.900,148.316
C08051=1212.258,279.635,-65.472,-176.714,6.897,148.317
C08052=1212.262,279.387,-65.444,-176.716,6.895,148.317
C08053=1212.266,279.139,-65.414,-176.718,6.892,148.317
C08054=1212.271,278.891,-65.387,-176.721,6.890,148.317
C08055=1212.275,278.642,-65.358,-176.723,6.888,148.317
C08056=1212.279,278.394,-65.330,-176.726,6.885,148.317
C08057=1212.284,278.145,-65.301,-176.728,6.883,148.317
C08058=1212.288,277.897,-65.273,-176.730,6.881,148.318
C08059=1212.293,277.648,-65.245,-176.733,6.878,148.318
C08060=1212.296,277.400,-65.217,-176.736,6.876,148.318
C08061=1212.301,277.152,-65.189,-176.738,6.873,148.318
C08062=1212.305,276.903,-65.160,-176.741,6.871,148.318
C08063=1212.310,276.655,-65.132,-176.743,6.869,148.318
C08064=1212.315,276.406,-65.105,-176.746,6.866,148.318
C08065=1212.319,276.158,-65.077,-176.748,6.864,148.319
C08066=1212.323,275.910,-65.049,-176.751,6.862,148.319
C08067=1212.328,275.661,-65.020,-176.753,6.859,148.319
C08068=1212.332,275.413,-64.992,-176.756,6.857,148.319
C08069=1212.336,275.165,-64.964,-176.758,6.855,148.319
C08070=1212.341,274.916,-64.936,-176.761,6.852,148.319
C08071=1212.345,274.668,-64.908,-176.763,6.850,148.319
C08072=1212.349,274.419,-64.881,-176.765,6.848,148.319
C08073=1212.354,274.170,-64.852,-176.769,6.845,148.320
C08074=1212.358,273.923,-64.824,-176.771,6.843,148.320
C08075=1212.362,273.675,-64.796,-176.773,6.841,148.320
C08076=1212.367,273.426,-64.768,-176.776,6.838,148.320
C08077=1212.372,273.177,-64.741,-176.778,6.836,148.320
C08078=1212.375,272.929,-64.712,-176.781,6.834,148.320
C08079=1212.380,272.681,-64.685,-176.783,6.831,148.320
C08080=1212.384,272.432,-64.656,-176.786,6.829,148.321
C08081=1212.389,272.183,-64.629,-176.788,6.827,148.321
C08082=1212.393,271.936,-64.601,-176.791,6.824,148.321
C08083=1212.397,271.687,-64.573,-176.794,6.822,148.321
C08084=1212.402,271.439,-64.544,-176.796,6.820,148.321
C08085=1212.406,271.190,-64.517,-176.799,6.817,148.322
C08086=1212.410,270.942,-64.489,-176.801,6.815,148.322
C08087=1212.415,270.694,-64.462,-176.803,6.812,148.322
C08088=1212.420,270.444,-64.433,-176.806,6.810,148.322
C08089=1212.424,270.196,-64.406,-176.808,6.808,148.322
C08090=1212.428,269.949,-64.378,-176.811,6.806,148.322
C08091=1212.432,269.699,-64.351,-176.814,6.803,148.322
C08092=1212.437,269.452,-64.323,-176.816,6.801,148.323
C08093=1212.441,269.203,-64.296,-176.818,6.799,148.323
C08094=1212.446,268.954,-64.267,-176.822,6.796,148.323
C08095=1212.450,268.706,-64.239,-176.824,6.794,148.323
C08096=1212.455,268.458,-64.212,-176.826,6.792,148.323
C08097=1212.459,268.209,-64.184,-176.829,6.789,148.323
C08098=1212.463,267.961,-64.157,-176.831,6.787,148.323
C08099=1212.468,267.713,-64.129,-176.834,6.785,148.324
C08100=1212.472,267.464,-64.102,-176.836,6.783,148.324
C08101=1212.477,267.215,-64.073,-176.839,6.780,148.324
C08102=1212.481,266.967,-64.046,-176.841,6.778,148.324
C08103=1212.485,266.718,-64.018,-176.844,6.776,148.324
C08104=1212.490,266.470,-63.991,-176.847,6.773,148.325
C08105=1212.494,266.222,-63.963,-176.849,6.771,148.325
C08106=1212.499,265.973,-63.936,-176.851,6.769,148.325
C08107=1212.503,265.724,-63.909,-176.854,6.766,148.325
C08108=1212.507,265.476,-63.881,-176.857,6.764,148.325
C08109=1212.512,265.228,-63.854,-176.859,6.762,148.326
C08110=1212.516,264.980,-63.826,-176.861,6.760,148.326
C08111=1212.520,264.731,-63.799,-176.864,6.757,148.326
C08112=1212.525,264.482,-63.772,-176.867,6.755,148.326
C08113=1212.529,264.234,-63.744,-176.869,6.753,148.326
C08114=1212.534,263.986,-63.717,-176.872,6.750,148.326
C08115=1212.538,263.737,-63.689,-176.874,6.748,148.326
C08116=1212.543,263.464,-63.659,-176.877,6.746,148.327
C08117=1212.548,263.192,-63.629,-176.880,6.743,148.327
C08118=1212.553,262.919,-63.599,-176.883,6.740,148.327
C08119=1212.557,262.646,-63.569,-176.885,6.738,148.327
C08120=1212.562,262.398,-63.542,-176.888,6.736,148.328
C08121=1212.566,262.149,-63.515,-176.890,6.733,148.328
C08122=1212.571,261.901,-63.487,-176.893,6.732,148.328
C08123=1212.575,261.653,-63.460,-176.895,6.729,148.328
C08124=1212.579,261.404,-63.433,-176.898,6.727,148.328
C08125=1212.584,261.155,-63.406,-176.901,6.724,148.328
C08126=1212.588,260.907,-63.378,-176.903,6.723,148.329
C08127=1212.593,260.659,-63.351,-176.905,6.720,148.329
C08128=1212.598,260.410,-63.324,-176.908,6.719,148.329
C08129=1212.602,260.161,-63.296,-176.911,6.716,148.329
C08130=1212.606,259.913,-63.270,-176.913,6.714,148.329
C08131=1212.610,259.664,-63.243,-176.915,6.711,148.329
C08132=1212.615,259.417,-63.215,-176.918,6.710,148.330
C08133=1212.619,259.168,-63.188,-176.921,6.707,148.330
C08134=1212.624,258.920,-63.161,-176.923,6.705,148.330
C08135=1212.628,258.670,-63.133,-176.926,6.703,148.330
C08136=1212.633,258.422,-63.106,-176.928,6.701,148.331
C08137=1212.637,258.174,-63.080,-176.931,6.698,148.331
C08138=1212.641,257.925,-63.053,-176.933,6.696,148.331
C08139=1212.646,257.677,-63.026,-176.936,6.694,148.331
C08140=1212.651,257.428,-62.999,-176.938,6.692,148.331
C08141=1212.655,257.180,-62.972,-176.941,6.689,148.332
C08142=1212.659,256.932,-62.945,-176.943,6.687,148.332
C08143=1212.663,256.682,-62.918,-176.946,6.685,148.332
C08144=1212.668,256.434,-62.891,-176.949,6.683,148.332
C08145=1212.673,256.185,-62.864,-176.951,6.680,148.332
C08146=1212.677,255.937,-62.837,-176.954,6.678,148.333
C08147=1212.681,255.689,-62.810,-176.956,6.676,148.333
C08148=1212.686,255.440,-62.783,-176.959,6.674,148.333
C08149=1212.690,255.192,-62.756,-176.961,6.672,148.333
C08150=1212.695,254.943,-62.729,-176.964,6.669,148.333
C08151=1212.699,254.695,-62.702,-176.967,6.667,148.334
C08152=1212.704,254.446,-62.675,-176.969,6.665,148.334
C08153=1212.708,254.198,-62.648,-176.971,6.663,148.334
C08154=1212.712,253.950,-62.622,-176.974,6.661,148.334
C08155=1212.717,253.700,-62.595,-176.977,6.658,148.334
C08156=1212.721,253.451,-62.568,-176.979,6.657,148.335
C08157=1212.725,253.203,-62.542,-176.981,6.654,148.335
C08158=1212.730,252.955,-62.515,-176.984,6.653,148.335
C08159=1212.734,252.706,-62.487,-176.986,6.650,148.335
C08160=1212.738,252.458,-62.461,-176.989,6.648,148.335
C08161=1212.743,252.209,-62.435,-176.992,6.645,148.336
C08162=1212.748,251.960,-62.408,-176.994,6.644,148.336
C08163=1212.752,251.712,-62.381,-176.997,6.642,148.336
C08164=1212.757,251.464,-62.354,-176.999,6.640,148.336
C08165=1212.761,251.215,-62.328,-177.002,6.637,148.336
C08166=1212.765,250.967,-62.301,-177.005,6.635,148.337
C08167=1212.770,250.718,-62.274,-177.007,6.633,148.337
C08168=1212.774,250.470,-62.248,-177.009,6.631,148.337
C08169=1212.779,250.221,-62.221,-177.012,6.629,148.337
C08170=1212.783,249.973,-62.195,-177.015,6.626,148.338
C08171=1212.788,249.724,-62.168,-177.017,6.624,148.338
C08172=1212.793,249.475,-62.141,-177.020,6.622,148.338
C08173=1212.796,249.227,-62.115,-177.022,6.620,148.338
C08174=1212.801,248.978,-62.088,-177.025,6.618,148.339
C08175=1212.805,248.729,-62.062,-177.027,6.616,148.339
C08176=1212.810,248.481,-62.035,-177.030,6.613,148.339
C08177=1212.814,248.233,-62.009,-177.032,6.611,148.339
C08178=1212.819,247.984,-61.982,-177.035,6.609,148.339
C08179=1212.823,247.736,-61.956,-177.037,6.608,148.340
C08180=1212.828,247.487,-61.930,-177.040,6.605,148.340
C08181=1212.832,247.239,-61.903,-177.043,6.603,148.340
C08182=1212.837,246.990,-61.877,-177.045,6.601,148.340
C08183=1212.841,246.742,-61.851,-177.048,6.599,148.340
C08184=1212.846,246.493,-61.824,-177.050,6.597,148.341
C08185=1212.850,246.244,-61.798,-177.053,6.595,148.341
C08186=1212.855,245.996,-61.771,-177.055,6.593,148.341
C08187=1212.859,245.747,-61.745,-177.058,6.591,148.341
C08188=1212.864,245.498,-61.718,-177.061,6.588,148.342
C08189=1212.868,245.250,-61.692,-177.063,6.586,148.342
C08190=1212.872,245.001,-61.666,-177.066,6.584,148.342
C08191=1212.877,244.753,-61.640,-177.068,6.582,148.342
C08192=1212.882,244.504,-61.614,-177.070,6.580,148.343
C08193=1212.886,244.256,-61.587,-177.073,6.578,148.343
C08194=1212.890,244.007,-61.561,-177.076,6.576,148.343
C08195=1212.894,243.759,-61.535,-177.078,6.573,148.343
C08196=1212.899,243.510,-61.508,-177.081,6.571,148.344
C08197=1212.903,243.261,-61.482,-177.083,6.570,148.344
C08198=1212.908,243.012,-61.456,-177.086,6.567,148.344
C08199=1212.913,242.764,-61.430,-177.088,6.566,148.344
C08200=1212.917,242.516,-61.404,-177.091,6.564,148.345
C08201=1212.922,242.267,-61.377,-177.093,6.562,148.345
C08202=1212.926,242.018,-61.352,-177.096,6.559,148.345
C08203=1212.930,241.770,-61.325,-177.099,6.557,148.345
C08204=1212.935,241.521,-61.299,-177.101,6.555,148.345
C08205=1212.940,241.273,-61.273,-177.104,6.553,148.346
C08206=1212.944,241.025,-61.247,-177.106,6.551,148.346
C08207=1212.949,240.775,-61.221,-177.109,6.549,148.346
C08208=1212.953,240.527,-61.195,-177.111,6.547,148.346
C08209=1212.957,240.278,-61.169,-177.114,6.545,148.347
C08210=1212.961,240.030,-61.143,-177.117,6.542,148.347
C08211=1212.967,239.781,-61.117,-177.119,6.540,148.347
C08212=1212.971,239.532,-61.091,-177.122,6.538,148.347
C08213=1212.975,239.284,-61.065,-177.124,6.537,148.348
C08214=1212.979,239.035,-61.039,-177.127,6.535,148.348
C08215=1212.985,238.787,-61.013,-177.129,6.533,148.348
C08216=1212.989,238.538,-60.987,-177.132,6.531,148.348
C08217=1212.993,238.289,-60.961,-177.134,6.529,148.349
C08218=1212.997,238.041,-60.935,-177.137,6.526,148.349
C08219=1213.002,237.791,-60.909,-177.140,6.524,148.349
C08220=1213.007,237.521,-60.881,-177.142,6.522,148.349
C08221=1213.012,237.249,-60.853,-177.145,6.520,148.350
C08222=1213.017,236.978,-60.825,-177.148,6.518,148.350
C08223=1213.022,236.707,-60.796,-177.151,6.516,148.350
C08224=1213.026,236.458,-60.770,-177.153,6.514,148.350
C08225=1213.031,236.210,-60.745,-177.155,6.512,148.351
C08226=1213.035,235.961,-60.719,-177.158,6.510,148.351
C08227=1213.040,235.712,-60.693,-177.161,6.507,148.351
C08228=1213.044,235.463,-60.667,-177.163,6.505,148.351
C08229=1213.049,235.215,-60.642,-177.166,6.503,148.352
C08230=1213.053,234.966,-60.616,-177.169,6.501,148.352
C08231=1213.057,234.717,-60.590,-177.171,6.499,148.352
C08232=1213.061,234.468,-60.565,-177.173,6.497,148.353
C08233=1213.066,234.220,-60.539,-177.176,6.495,148.353
C08234=1213.071,233.971,-60.513,-177.179,6.494,148.353
C08235=1213.076,233.722,-60.487,-177.181,6.492,148.354
C08236=1213.080,233.474,-60.462,-177.183,6.489,148.354
C08237=1213.085,233.225,-60.436,-177.186,6.488,148.354
C08238=1213.089,232.977,-60.410,-177.189,6.485,148.354
C08239=1213.094,232.729,-60.385,-177.192,6.483,148.355
C08240=1213.098,232.480,-60.359,-177.194,6.481,148.355
C08241=1213.102,232.230,-60.334,-177.197,6.479,148.355
C08242=1213.107,231.982,-60.309,-177.199,6.477,148.355
C08243=1213.111,231.733,-60.283,-177.202,6.475,148.356
C08244=1213.116,231.485,-60.257,-177.204,6.473,148.356
C08245=1213.120,231.237,-60.232,-177.207,6.471,148.356
C08246=1213.125,230.988,-60.206,-177.209,6.469,148.356
C08247=1213.130,230.740,-60.181,-177.212,6.468,148.357
C08248=1213.134,230.490,-60.156,-177.215,6.466,148.357
C08249=1213.138,230.241,-60.130,-177.217,6.464,148.357
C08250=1213.143,229.993,-60.104,-177.219,6.462,148.357
C08251=1213.147,229.744,-60.079,-177.222,6.460,148.358
C08252=1213.152,229.495,-60.054,-177.225,6.458,148.358
C08253=1213.157,229.247,-60.028,-177.228,6.455,148.358
C08254=1213.161,228.998,-60.003,-177.230,6.453,148.358
C08255=1213.166,228.750,-59.977,-177.233,6.451,148.359
C08256=1213.170,228.501,-59.952,-177.235,6.449,148.359
C08257=1213.174,228.252,-59.926,-177.238,6.448,148.359
C08258=1213.179,228.004,-59.902,-177.240,6.446,148.360
C08259=1213.183,227.755,-59.876,-177.243,6.444,148.360
C08260=1213.188,227.506,-59.851,-177.245,6.442,148.360
C08261=1213.192,227.258,-59.825,-177.248,6.440,148.361
C08262=1213.197,227.010,-59.800,-177.250,6.438,148.361
C08263=1213.202,226.760,-59.775,-177.253,6.436,148.361
C08264=1213.206,226.511,-59.749,-177.256,6.434,148.361
C08265=1213.211,226.263,-59.725,-177.258,6.432,148.362
C08266=1213.215,226.014,-59.699,-177.261,6.430,148.362
C08267=1213.219,225.766,-59.674,-177.263,6.428,148.362
C08268=1213.224,225.517,-59.649,-177.266,6.427,148.363
C08269=1213.229,225.268,-59.624,-177.268,6.425,148.363
C08270=1213.233,225.019,-59.599,-177.271,6.423,148.363
C08271=1213.238,224.771,-59.573,-177.273,6.421,148.363
C08272=1213.242,224.522,-59.548,-177.276,6.419,148.364
C08273=1213.247,224.274,-59.523,-177.278,6.417,148.364
C08274=1213.251,224.024,-59.498,-177.282,6.414,148.364
C08275=1213.256,223.776,-59.473,-177.284,6.413,148.365
C08276=1213.260,223.527,-59.448,-177.287,6.411,148.365
C08277=1213.265,223.279,-59.423,-177.289,6.408,148.365
C08278=1213.269,223.030,-59.398,-177.292,6.407,148.365
C08279=1213.274,222.781,-59.373,-177.294,6.405,148.366
C08280=1213.278,222.532,-59.348,-177.297,6.403,148.366
C08281=1213.283,222.284,-59.322,-177.300,6.401,148.366
C08282=1213.287,222.035,-59.298,-177.302,6.399,148.367
C08283=1213.292,221.787,-59.272,-177.305,6.397,148.367
C08284=1213.296,221.537,-59.247,-177.307,6.395,148.367
C08285=1213.301,221.289,-59.223,-177.310,6.393,148.367
C08286=1213.305,221.040,-59.198,-177.312,6.392,148.368
C08287=1213.310,220.791,-59.173,-177.315,6.390,148.368
C08288=1213.314,220.543,-59.147,-177.318,6.388,148.368
C08289=1213.319,220.294,-59.123,-177.320,6.386,148.369
C08290=1213.324,220.045,-59.098,-177.323,6.384,148.369
C08291=1213.328,219.797,-59.073,-177.325,6.382,148.369
C08292=1213.332,219.548,-59.049,-177.328,6.380,148.370
C08293=1213.337,219.299,-59.024,-177.330,6.378,148.370
C08294=1213.342,219.051,-58.998,-177.333,6.376,148.370
C08295=1213.346,218.802,-58.974,-177.336,6.375,148.371
C08296=1213.351,218.553,-58.949,-177.338,6.373,148.371
C08297=1213.355,218.304,-58.925,-177.341,6.371,148.371
C08298=1213.359,218.056,-58.899,-177.343,6.369,148.371
C08299=1213.365,217.807,-58.875,-177.346,6.367,148.372
C08300=1213.368,217.558,-58.850,-177.348,6.365,148.372
C08301=1213.373,217.309,-58.825,-177.351,6.363,148.372
C08302=1213.378,217.061,-58.801,-177.353,6.361,148.373
C08303=1213.382,216.812,-58.776,-177.356,6.359,148.373
C08304=1213.387,216.563,-58.751,-177.359,6.358,148.373
C08305=1213.392,216.315,-58.727,-177.361,6.356,148.374
C08306=1213.396,216.065,-58.702,-177.364,6.354,148.374
C08307=1213.400,215.818,-58.677,-177.367,6.352,148.374
C08308=1213.405,215.568,-58.652,-177.369,6.350,148.375
C08309=1213.409,215.320,-58.628,-177.372,6.348,148.375
C08310=1213.414,215.071,-58.603,-177.375,6.347,148.375
C08311=1213.418,214.822,-58.579,-177.377,6.344,148.375
C08312=1213.423,214.573,-58.554,-177.379,6.343,148.376
C08313=1213.428,214.325,-58.530,-177.382,6.341,148.376
C08314=1213.432,214.075,-58.505,-177.385,6.339,148.376
C08315=1213.436,213.827,-58.481,-177.387,6.337,148.377
C08316=1213.442,213.578,-58.456,-177.390,6.335,148.377
C08317=1213.445,213.329,-58.432,-177.393,6.333,148.377
C08318=1213.451,213.080,-58.407,-177.395,6.332,148.378
C08319=1213.455,212.833,-58.382,-177.398,6.330,148.378
C08320=1213.460,212.584,-58.358,-177.400,6.328,148.378
C08321=1213.464,212.335,-58.333,-177.403,6.326,148.379
C08322=1213.469,212.086,-58.309,-177.406,6.324,148.379
C08323=1213.473,211.838,-58.285,-177.408,6.322,148.379
C08324=1213.478,211.566,-58.258,-177.411,6.320,148.380
C08325=1213.483,211.296,-58.232,-177.414,6.319,148.380
C08326=1213.488,211.026,-58.205,-177.417,6.316,148.380
C08327=1213.493,210.756,-58.179,-177.420,6.314,148.381
C08328=1213.498,210.506,-58.155,-177.422,6.312,148.381
C08329=1213.502,210.257,-58.130,-177.425,6.310,148.381
C08330=1213.507,210.009,-58.106,-177.427,6.309,148.382
C08331=1213.511,209.760,-58.082,-177.430,6.307,148.382
C08332=1213.516,209.512,-58.057,-177.433,6.305,148.382
C08333=1213.520,209.262,-58.032,-177.435,6.304,148.383
C08334=1213.525,209.014,-58.008,-177.437,6.302,148.383
C08335=1213.529,208.766,-57.984,-177.440,6.300,148.383
C08336=1213.535,208.516,-57.960,-177.443,6.298,148.384
C08337=1213.538,208.267,-57.936,-177.445,6.297,148.384
C08338=1213.543,208.019,-57.912,-177.448,6.295,148.384
C08339=1213.548,207.770,-57.887,-177.450,6.293,148.385
C08340=1213.552,207.522,-57.863,-177.453,6.291,148.385
C08341=1213.557,207.273,-57.840,-177.455,6.289,148.385
C08342=1213.562,207.023,-57.815,-177.458,6.287,148.386
C08343=1213.566,206.775,-57.791,-177.461,6.285,148.386
C08344=1213.570,206.526,-57.767,-177.463,6.283,148.386
C08345=1213.576,206.277,-57.743,-177.466,6.282,148.387
C08346=1213.580,206.029,-57.719,-177.469,6.280,148.387
C08347=1213.584,205.779,-57.694,-177.471,6.278,148.387
C08348=1213.588,205.531,-57.670,-177.474,6.276,148.388
C08349=1213.594,205.282,-57.646,-177.477,6.274,148.388
C08350=1213.598,205.033,-57.622,-177.479,6.273,148.388
C08351=1213.603,204.785,-57.598,-177.481,6.271,148.389
C08352=1213.607,204.536,-57.575,-177.484,6.269,148.389
C08353=1213.612,204.286,-57.549,-177.487,6.268,148.389
C08354=1213.616,204.038,-57.525,-177.489,6.266,148.390
C08355=1213.621,203.789,-57.502,-177.492,6.264,148.390
C08356=1213.625,203.541,-57.478,-177.495,6.262,148.390
C08357=1213.630,203.291,-57.455,-177.497,6.260,148.391
C08358=1213.634,203.043,-57.431,-177.500,6.258,148.391
C08359=1213.639,202.794,-57.406,-177.502,6.257,148.391
C08360=1213.644,202.545,-57.382,-177.505,6.255,148.392
C08361=1213.648,202.296,-57.358,-177.508,6.253,148.392
C08362=1213.653,202.047,-57.335,-177.510,6.252,148.392
C08363=1213.657,201.799,-57.311,-177.512,6.250,148.393
C08364=1213.662,201.550,-57.287,-177.515,6.248,148.393
C08365=1213.667,201.301,-57.263,-177.518,6.246,148.393
C08366=1213.672,201.052,-57.239,-177.520,6.245,148.394
C08367=1213.676,200.804,-57.215,-177.523,6.243,148.394
C08368=1213.681,200.555,-57.192,-177.526,6.241,148.394
C08369=1213.685,200.306,-57.168,-177.528,6.239,148.395
C08370=1213.690,200.057,-57.144,-177.531,6.237,148.395
C08371=1213.694,199.808,-57.120,-177.534,6.235,148.395
C08372=1213.698,199.559,-57.097,-177.536,6.234,148.396
C08373=1213.703,199.311,-57.073,-177.538,6.233,148.396
C08374=1213.707,199.061,-57.049,-177.541,6.231,148.397
C08375=1213.712,198.812,-57.026,-177.544,6.229,148.397
C08376=1213.716,198.564,-57.002,-177.546,6.227,148.397
C08377=1213.721,198.315,-56.978,-177.549,6.225,148.398
C08378=1213.726,198.066,-56.954,-177.552,6.223,148.398
C08379=1213.731,197.817,-56.930,-177.554,6.222,148.398
C08380=1213.736,197.568,-56.907,-177.557,6.220,148.399
C08381=1213.740,197.320,-56.883,-177.559,6.219,148.399
C08382=1213.745,197.071,-56.860,-177.562,6.217,148.399
C08383=1213.749,196.822,-56.836,-177.564,6.215,148.400
C08384=1213.754,196.573,-56.812,-177.567,6.213,148.400
C08385=1213.759,196.324,-56.789,-177.570,6.212,148.401
C08386=1213.763,196.075,-56.765,-177.573,6.210,148.401
C08387=1213.768,195.827,-56.741,-177.575,6.208,148.401
C08388=1213.772,195.578,-56.719,-177.578,6.206,148.402
C08389=1213.776,195.329,-56.695,-177.580,6.205,148.402
C08390=1213.781,195.080,-56.672,-177.583,6.203,148.402
C08391=1213.785,194.832,-56.648,-177.585,6.202,148.403
C08392=1213.790,194.583,-56.624,-177.588,6.200,148.403
C08393=1213.795,194.334,-56.601,-177.591,6.198,148.403
C08394=1213.800,194.085,-56.578,-177.593,6.196,148.404
C08395=1213.804,193.836,-56.554,-177.596,6.194,148.404
C08396=1213.809,193.587,-56.530,-177.598,6.193,148.404
C08397=1213.813,193.338,-56.507,-177.601,6.191,148.405
C08398=1213.818,193.089,-56.484,-177.603,6.190,148.405
C08399=1213.823,192.840,-56.460,-177.606,6.188,148.405
C08400=1213.827,192.591,-56.437,-177.609,6.186,148.406
C08401=1213.831,192.342,-56.414,-177.611,6.184,148.406
C08402=1213.836,192.095,-56.390,-177.613,6.183,148.407
C08403=1213.841,191.846,-56.367,-177.616,6.181,148.407
C08404=1213.846,191.597,-56.344,-177.619,6.180,148.407
C08405=1213.850,191.347,-56.320,-177.622,6.178,148.408
C08406=1213.855,191.098,-56.297,-177.624,6.176,148.408
C08407=1213.859,190.850,-56.274,-177.627,6.174,148.409
C08408=1213.864,190.601,-56.251,-177.629,6.173,148.409
C08409=1213.869,190.352,-56.227,-177.632,6.171,148.409
C08410=1213.873,190.103,-56.204,-177.635,6.170,148.410
C08411=1213.878,189.854,-56.181,-177.637,6.168,148.410
C08412=1213.883,189.605,-56.157,-177.640,6.166,148.410
C08413=1213.887,189.357,-56.135,-177.642,6.164,148.411
C08414=1213.892,189.107,-56.112,-177.645,6.163,148.411
C08415=1213.897,188.858,-56.088,-177.647,6.161,148.411
C08416=1213.901,188.609,-56.065,-177.650,6.160,148.412
C08417=1213.905,188.361,-56.042,-177.653,6.158,148.412
C08418=1213.910,188.112,-56.019,-177.656,6.156,148.413
C08419=1213.915,187.863,-55.995,-177.658,6.155,148.413
C08420=1213.920,187.614,-55.972,-177.660,6.153,148.413
C08421=1213.924,187.366,-55.950,-177.663,6.152,148.414
C08422=1213.929,187.117,-55.926,-177.666,6.150,148.414
C08423=1213.933,186.868,-55.903,-177.668,6.148,148.414
C08424=1213.938,186.618,-55.880,-177.671,6.146,148.415
C08425=1213.942,186.369,-55.858,-177.673,6.145,148.415
C08426=1213.948,186.121,-55.835,-177.676,6.143,148.416
C08427=1213.952,185.872,-55.811,-177.679,6.142,148.416
C08428=1213.957,185.602,-55.787,-177.682,6.140,148.416
C08429=1213.962,185.333,-55.762,-177.684,6.138,148.417
C08430=1213.967,185.063,-55.737,-177.687,6.136,148.417
C08431=1213.972,184.793,-55.712,-177.690,6.135,148.418
C08432=1213.977,184.544,-55.689,-177.693,6.133,148.418
C08433=1213.981,184.296,-55.666,-177.695,6.131,148.418
C08434=1213.985,184.047,-55.643,-177.697,6.130,148.419
C08435=1213.990,183.798,-55.619,-177.700,6.128,148.419
C08436=1213.995,183.549,-55.598,-177.703,6.127,148.420
C08437=1214.000,183.300,-55.574,-177.705,6.125,148.420
C08438=1214.004,183.051,-55.552,-177.708,6.123,148.420
C08439=1214.008,182.802,-55.528,-177.711,6.122,148.421
C08440=1214.014,182.553,-55.506,-177.713,6.120,148.421
C08441=1214.018,182.304,-55.483,-177.716,6.119,148.422
C08442=1214.023,182.055,-55.460,-177.719,6.117,148.422
C08443=1214.027,181.806,-55.438,-177.721,6.116,148.422
C08444=1214.032,181.558,-55.415,-177.723,6.114,148.423
C08445=1214.036,181.309,-55.392,-177.726,6.112,148.423
C08446=1214.041,181.059,-55.369,-177.729,6.111,148.424
C08447=1214.046,180.810,-55.346,-177.732,6.109,148.424
C08448=1214.050,180.562,-55.324,-177.734,6.108,148.424
C08449=1214.055,180.313,-55.301,-177.736,6.106,148.425
C08450=1214.059,180.064,-55.278,-177.739,6.104,148.425
C08451=1214.064,179.814,-55.256,-177.742,6.102,148.425
C08452=1214.069,179.566,-55.233,-177.744,6.101,148.426
C08453=1214.074,179.317,-55.210,-177.747,6.100,148.426
C08454=1214.078,179.068,-55.188,-177.750,6.098,148.427
C08455=1214.083,178.820,-55.165,-177.752,6.096,148.427
C08456=1214.088,178.570,-55.143,-177.754,6.095,148.427
C08457=1214.092,178.321,-55.119,-177.757,6.093,148.428
C08458=1214.097,178.073,-55.098,-177.760,6.092,148.428
C08459=1214.101,177.824,-55.075,-177.762,6.090,148.428
C08460=1214.106,177.574,-55.052,-177.765,6.089,148.429
C08461=1214.111,177.326,-55.030,-177.768,6.087,148.429
C08462=1214.116,177.076,-55.007,-177.770,6.085,148.430
C08463=1214.120,176.828,-54.984,-177.773,6.084,148.430
C08464=1214.125,176.579,-54.962,-177.775,6.083,148.431
C08465=1214.129,176.330,-54.939,-177.778,6.081,148.431
C08466=1214.133,176.081,-54.917,-177.781,6.079,148.432
C08467=1214.139,175.832,-54.894,-177.783,6.078,148.432
C08468=1214.143,175.583,-54.872,-177.786,6.077,148.432
C08469=1214.148,175.334,-54.849,-177.788,6.075,148.433
C08470=1214.153,175.085,-54.827,-177.791,6.073,148.433
C08471=1214.157,174.836,-54.805,-177.793,6.072,148.433
C08472=1214.162,174.588,-54.782,-177.796,6.070,148.434
C08473=1214.166,174.338,-54.760,-177.799,6.069,148.434
C08474=1214.171,174.089,-54.738,-177.801,6.067,148.435
C08475=1214.176,173.841,-54.715,-177.804,6.066,148.435
C08476=1214.180,173.591,-54.693,-177.806,6.064,148.435
C08477=1214.185,173.342,-54.670,-177.809,6.062,148.436
C08478=1214.190,173.094,-54.648,-177.811,6.062,148.436
C08479=1214.194,172.844,-54.626,-177.814,6.060,148.437
C08480=1214.199,172.596,-54.604,-177.817,6.058,148.437
C08481=1214.204,172.347,-54.581,-177.819,6.056,148.437
C08482=1214.209,172.098,-54.559,-177.822,6.055,148.438
C08483=1214.213,171.849,-54.537,-177.825,6.054,148.438
C08484=1214.218,171.599,-54.515,-177.827,6.052,148.439
C08485=1214.222,171.351,-54.492,-177.829,6.051,148.439
C08486=1214.227,171.102,-54.470,-177.832,6.049,148.440
C08487=1214.232,170.853,-54.448,-177.835,6.047,148.440
C08488=1214.237,170.603,-54.426,-177.838,6.046,148.440
C08489=1214.241,170.355,-54.403,-177.840,6.045,148.441
C08490=1214.245,170.106,-54.381,-177.843,6.043,148.441
C08491=1214.250,169.857,-54.360,-177.845,6.041,148.442
C08492=1214.255,169.608,-54.337,-177.848,6.040,148.442
C08493=1214.260,169.359,-54.315,-177.851,6.039,148.443
C08494=1214.264,169.110,-54.293,-177.853,6.037,148.443
C08495=1214.268,168.861,-54.271,-177.855,6.036,148.443
C08496=1214.274,168.612,-54.248,-177.858,6.034,148.444
C08497=1214.278,168.363,-54.226,-177.861,6.032,148.444
C08498=1214.283,168.114,-54.205,-177.863,6.032,148.445
C08499=1214.287,167.865,-54.183,-177.866,6.030,148.445
C08500=1214.292,167.616,-54.161,-177.869,6.028,148.445
C08501=1214.296,167.367,-54.139,-177.871,6.027,148.446
C08502=1214.302,167.118,-54.117,-177.874,6.025,148.446
C08503=1214.306,166.869,-54.094,-177.876,6.024,148.447
C08504=1214.311,166.620,-54.072,-177.879,6.022,148.447
C08505=1214.316,166.372,-54.050,-177.881,6.021,148.447
C08506=1214.320,166.123,-54.028,-177.884,6.019,148.448
C08507=1214.325,165.874,-54.007,-177.887,6.018,148.448
C08508=1214.329,165.625,-53.985,-177.889,6.017,148.449
C08509=1214.334,165.376,-53.963,-177.892,6.015,148.449
C08510=1214.339,165.126,-53.940,-177.895,6.013,148.450
C08511=1214.344,164.878,-53.919,-177.897,6.012,148.450
C08512=1214.348,164.628,-53.897,-177.900,6.010,148.451
C08513=1214.353,164.380,-53.875,-177.902,6.009,148.451
C08514=1214.357,164.130,-53.853,-177.905,6.008,148.452
C08515=1214.363,163.881,-53.832,-177.908,6.006,148.452
C08516=1214.367,163.632,-53.810,-177.910,6.005,148.452
C08517=1214.372,163.383,-53.788,-177.912,6.003,148.453
C08518=1214.377,163.134,-53.766,-177.915,6.002,148.453
C08519=1214.381,162.885,-53.744,-177.918,6.001,148.454
C08520=1214.386,162.636,-53.723,-177.920,5.999,148.454
C08521=1214.390,162.387,-53.701,-177.923,5.997,148.454
C08522=1214.395,162.138,-53.679,-177.926,5.997,148.455
C08523=1214.400,161.890,-53.657,-177.928,5.995,148.455
C08524=1214.404,161.640,-53.636,-177.931,5.993,148.456
C08525=1214.409,161.391,-53.614,-177.933,5.992,148.456
C08526=1214.413,161.142,-53.592,-177.936,5.991,148.457
C08527=1214.418,160.893,-53.571,-177.939,5.989,148.457
C08528=1214.423,160.645,-53.549,-177.941,5.988,148.457
C08529=1214.427,160.395,-53.527,-177.944,5.986,148.458
C08530=1214.433,160.146,-53.506,-177.946,5.985,148.458
C08531=1214.437,159.897,-53.484,-177.949,5.984,148.459
C08532=1214.443,159.628,-53.461,-177.952,5.982,148.459
C08533=1214.447,159.360,-53.437,-177.955,5.980,148.460
C08534=1214.453,159.090,-53.414,-177.957,5.978,148.460
C08535=1214.458,158.821,-53.391,-177.960,5.978,148.461
C08536=1214.462,158.572,-53.369,-177.963,5.976,148.461
C08537=1214.467,158.323,-53.347,-177.965,5.974,148.461
C08538=1214.472,158.075,-53.326,-177.968,5.974,148.462
C08539=1214.476,157.825,-53.304,-177.971,5.972,148.462
C08540=1214.481,157.576,-53.283,-177.973,5.970,148.463
C08541=1214.486,157.327,-53.261,-177.975,5.969,148.463
C08542=1214.490,157.077,-53.240,-177.978,5.967,148.464
C08543=1214.495,156.829,-53.218,-177.981,5.966,148.464
C08544=1214.499,156.580,-53.197,-177.983,5.965,148.465
C08545=1214.504,156.330,-53.176,-177.986,5.963,148.465
C08546=1214.509,156.082,-53.154,-177.988,5.962,148.466
C08547=1214.514,155.832,-53.133,-177.991,5.960,148.466
C08548=1214.518,155.583,-53.111,-177.993,5.959,148.466
C08549=1214.523,155.334,-53.089,-177.996,5.958,148.467
C08550=1214.528,155.085,-53.068,-177.999,5.956,148.467
C08551=1214.533,154.837,-53.047,-178.001,5.955,148.468
C08552=1214.537,154.587,-53.026,-178.004,5.954,148.468
C08553=1214.542,154.338,-53.004,-178.006,5.953,148.469
C08554=1214.547,154.089,-52.983,-178.009,5.951,148.469
C08555=1214.552,153.840,-52.962,-178.012,5.949,148.470
C08556=1214.556,153.591,-52.940,-178.014,5.949,148.470
C08557=1214.561,153.342,-52.919,-178.017,5.947,148.470
C08558=1214.566,153.093,-52.897,-178.019,5.946,148.471
C08559=1214.571,152.844,-52.876,-178.022,5.944,148.471
C08560=1214.574,152.595,-52.855,-178.025,5.942,148.472
C08561=1214.579,152.346,-52.834,-178.027,5.941,148.472
C08562=1214.585,152.097,-52.813,-178.030,5.940,148.473
C08563=1214.590,151.848,-52.791,-178.032,5.939,148.473
C08564=1214.593,151.598,-52.771,-178.035,5.937,148.474
C08565=1214.598,151.350,-52.749,-178.038,5.937,148.474
C08566=1214.603,151.100,-52.728,-178.040,5.935,148.475
C08567=1214.608,150.852,-52.706,-178.043,5.933,148.475
C08568=1214.613,150.603,-52.686,-178.046,5.932,148.476
C08569=1214.617,150.353,-52.665,-178.048,5.931,148.476
C08570=1214.622,150.104,-52.643,-178.050,5.930,148.476
C08571=1214.627,149.855,-52.623,-178.053,5.928,148.477
C08572=1214.631,149.607,-52.601,-178.056,5.927,148.477
C08573=1214.637,149.357,-52.580,-178.058,5.925,148.478
C08574=1214.641,149.108,-52.560,-178.061,5.924,148.478
C08575=1214.645,148.859,-52.538,-178.064,5.923,148.479
C08576=1214.651,148.610,-52.517,-178.066,5.921,148.479
C08577=1214.655,148.361,-52.496,-178.069,5.920,148.480
C08578=1214.660,148.112,-52.474,-178.071,5.919,148.480
C08579=1214.665,147.863,-52.454,-178.074,5.918,148.481
C08580=1214.669,147.614,-52.433,-178.077,5.916,148.481
C08581=1214.674,147.364,-52.412,-178.079,5.915,148.482
C08582=1214.678,147.116,-52.391,-178.082,5.913,148.482
C08583=1214.683,146.867,-52.370,-178.085,5.912,148.482
C08584=1214.688,146.617,-52.349,-178.087,5.911,148.483
C08585=1214.693,146.368,-52.328,-178.089,5.909,148.483
C08586=1214.698,146.120,-52.307,-178.092,5.909,148.484
C08587=1214.702,145.871,-52.286,-178.095,5.907,148.484
C08588=1214.707,145.621,-52.265,-178.097,5.906,148.485
C08589=1214.711,145.372,-52.245,-178.100,5.904,148.485
C08590=1214.716,145.123,-52.224,-178.102,5.903,148.486
C08591=1214.721,144.874,-52.202,-178.105,5.902,148.486
C08592=1214.726,144.625,-52.182,-178.107,5.901,148.487
C08593=1214.731,144.376,-52.161,-178.110,5.899,148.487
C08594=1214.735,144.127,-52.140,-178.113,5.899,148.488
C08595=1214.740,143.878,-52.119,-178.115,5.897,148.488
C08596=1214.745,143.629,-52.099,-178.118,5.895,148.488
C08597=1214.750,143.379,-52.078,-178.121,5.894,148.489
C08598=1214.754,143.131,-52.057,-178.123,5.893,148.489
C08599=1214.759,142.881,-52.036,-178.125,5.892,148.490
C08600=1214.763,142.632,-52.015,-178.129,5.890,148.490
C08601=1214.768,142.383,-51.994,-178.131,5.889,148.491
C08602=1214.773,142.134,-51.974,-178.134,5.888,148.491
C08603=1214.778,141.885,-51.953,-178.136,5.887,148.492
C08604=1214.782,141.636,-51.933,-178.139,5.885,148.492
C08605=1214.787,141.387,-51.912,-178.141,5.884,148.493
C08606=1214.792,141.137,-51.891,-178.144,5.882,148.493
C08607=1214.797,140.888,-51.871,-178.146,5.881,148.494
C08608=1214.802,140.639,-51.850,-178.149,5.880,148.494
C08609=1214.806,140.390,-51.829,-178.151,5.879,148.495
C08610=1214.811,140.141,-51.809,-178.154,5.878,148.495
C08611=1214.816,139.892,-51.788,-178.157,5.877,148.496
C08612=1214.820,139.643,-51.768,-178.159,5.875,148.496
C08613=1214.825,139.394,-51.747,-178.162,5.874,148.497
C08614=1214.830,139.145,-51.726,-178.165,5.872,148.497
C08615=1214.835,138.896,-51.705,-178.167,5.872,148.498
C08616=1214.839,138.647,-51.685,-178.170,5.870,148.498
C08617=1214.844,138.398,-51.665,-178.172,5.869,148.498
C08618=1214.849,138.149,-51.644,-178.175,5.868,148.499
C08619=1214.853,137.900,-51.623,-178.177,5.867,148.499
C08620=1214.858,137.650,-51.604,-178.180,5.865,148.500
C08621=1214.863,137.401,-51.583,-178.182,5.864,148.500
C08622=1214.868,137.152,-51.562,-178.185,5.862,148.501
C08623=1214.872,136.903,-51.542,-178.188,5.862,148.501
C08624=1214.877,136.654,-51.521,-178.190,5.860,148.502
C08625=1214.882,136.405,-51.501,-178.193,5.859,148.503
C08626=1214.886,136.156,-51.480,-178.196,5.858,148.503
C08627=1214.892,135.906,-51.460,-178.198,5.857,148.503
C08628=1214.896,135.657,-51.440,-178.201,5.855,148.504
C08629=1214.901,135.408,-51.419,-178.203,5.854,148.504
C08630=1214.906,135.159,-51.398,-178.206,5.853,148.505
C08631=1214.910,134.910,-51.378,-178.208,5.852,148.505
C08632=1214.915,134.660,-51.358,-178.212,5.850,148.506
C08633=1214.920,134.412,-51.338,-178.214,5.849,148.506
C08634=1214.925,134.163,-51.317,-178.216,5.848,148.507
C08635=1214.930,133.914,-51.297,-178.219,5.847,148.507
C08636=1214.935,133.645,-51.275,-178.222,5.845,148.508
C08637=1214.939,133.376,-51.253,-178.224,5.845,148.508
C08638=1214.945,133.107,-51.231,-178.227,5.843,148.509
C08639=1214.950,132.839,-51.210,-178.230,5.841,148.509
C08640=1214.955,132.589,-51.189,-178.233,5.841,148.510
C08641=1214.959,132.340,-51.169,-178.235,5.839,148.510
C08642=1214.964,132.091,-51.149,-178.238,5.838,148.511
C08643=1214.969,131.842,-51.129,-178.240,5.837,148.511
C08644=1214.974,131.593,-51.108,-178.243,5.835,148.512
C08645=1214.979,131.344,-51.088,-178.245,5.835,148.512
C08646=1214.984,131.095,-51.068,-178.248,5.833,148.513
C08647=1214.988,130.846,-51.048,-178.251,5.832,148.513
C08648=1214.993,130.597,-51.028,-178.253,5.831,148.514
C08649=1214.997,130.347,-51.008,-178.256,5.830,148.514
C08650=1215.002,130.098,-50.987,-178.259,5.828,148.515
C08651=1215.008,129.849,-50.968,-178.261,5.828,148.515
C08652=1215.012,129.600,-50.947,-178.263,5.827,148.516
C08653=1215.017,129.350,-50.928,-178.266,5.825,148.516
C08654=1215.021,129.101,-50.907,-178.269,5.824,148.517
C08655=1215.026,128.853,-50.887,-178.271,5.822,148.517
C08656=1215.031,128.603,-50.867,-178.274,5.822,148.518
C08657=1215.036,128.355,-50.847,-178.277,5.820,148.518
C08658=1215.041,128.105,-50.827,-178.279,5.819,148.519
C08659=1215.046,127.856,-50.807,-178.282,5.818,148.519
C08660=1215.050,127.606,-50.787,-178.284,5.817,148.520
C08661=1215.055,127.357,-50.767,-178.287,5.816,148.520
C08662=1215.059,127.108,-50.747,-178.290,5.815,148.521
C08663=1215.064,126.860,-50.727,-178.292,5.814,148.521
C08664=1215.069,126.610,-50.707,-178.295,5.812,148.522
C08665=1215.074,126.361,-50.687,-178.297,5.811,148.522
C08666=1215.078,126.111,-50.667,-178.299,5.810,148.523
C08667=1215.084,125.863,-50.648,-178.302,5.809,148.523
C08668=1215.088,125.614,-50.628,-178.305,5.808,148.524
C08669=1215.093,125.364,-50.608,-178.308,5.806,148.524
C08670=1215.097,125.115,-50.588,-178.310,5.806,148.525
C08671=1215.102,124.866,-50.568,-178.313,5.804,148.526
C08672=1215.107,124.617,-50.549,-178.315,5.803,148.526
C08673=1215.112,124.368,-50.528,-178.318,5.803,148.527
C08674=1215.117,124.118,-50.509,-178.320,5.801,148.527
C08675=1215.121,123.869,-50.488,-178.323,5.800,148.528
C08676=1215.126,123.620,-50.469,-178.326,5.798,148.528
C08677=1215.131,123.371,-50.449,-178.328,5.798,148.529
C08678=1215.136,123.122,-50.429,-178.330,5.797,148.529
C08679=1215.140,122.872,-50.409,-178.334,5.795,148.530
C08680=1215.146,122.623,-50.390,-178.336,5.794,148.530
C08681=1215.150,122.374,-50.370,-178.339,5.793,148.531
C08682=1215.155,122.125,-50.350,-178.341,5.792,148.531
C08683=1215.160,121.876,-50.331,-178.344,5.791,148.532
C08684=1215.165,121.626,-50.311,-178.346,5.790,148.532
C08685=1215.169,121.378,-50.291,-178.349,5.789,148.533
C08686=1215.174,121.128,-50.271,-178.352,5.787,148.533
C08687=1215.179,120.879,-50.252,-178.354,5.787,148.534
C08688=1215.183,120.630,-50.233,-178.356,5.786,148.534
C08689=1215.188,120.381,-50.212,-178.360,5.784,148.535
C08690=1215.193,120.132,-50.193,-178.362,5.783,148.535
C08691=1215.198,119.882,-50.173,-178.365,5.782,148.536
C08692=1215.203,119.633,-50.154,-178.367,5.781,148.536
C08693=1215.208,119.384,-50.134,-178.370,5.780,148.537
C08694=1215.213,119.135,-50.114,-178.372,5.778,148.537
C08695=1215.217,118.885,-50.094,-178.375,5.778,148.538
C08696=1215.222,118.637,-50.076,-178.377,5.777,148.538
C08697=1215.227,118.387,-50.056,-178.380,5.775,148.539
C08698=1215.231,118.138,-50.036,-178.382,5.774,148.539
C08699=1215.237,117.889,-50.017,-178.385,5.773,148.540
C08700=1215.241,117.639,-49.997,-178.388,5.772,148.540
C08701=1215.246,117.390,-49.977,-178.390,5.771,148.541
C08702=1215.250,117.142,-49.958,-178.393,5.770,148.541
C08703=1215.255,116.892,-49.939,-178.395,5.769,148.542
C08704=1215.260,116.643,-49.919,-178.398,5.768,148.542
C08705=1215.265,116.394,-49.900,-178.401,5.767,148.543
C08706=1215.270,116.144,-49.880,-178.403,5.766,148.544
C08707=1215.275,115.896,-49.861,-178.405,5.765,148.544
C08708=1215.279,115.646,-49.842,-178.408,5.763,148.545
C08709=1215.284,115.397,-49.822,-178.411,5.763,148.545
C08710=1215.290,115.148,-49.803,-178.413,5.761,148.546
C08711=1215.294,114.898,-49.784,-178.416,5.760,148.546
C08712=1215.299,114.650,-49.764,-178.418,5.759,148.547
C08713=1215.304,114.400,-49.745,-178.421,5.758,148.547
C08714=1215.308,114.150,-49.725,-178.423,5.757,148.548
C08715=1215.313,113.902,-49.706,-178.426,5.756,148.548
C08716=1215.318,113.652,-49.687,-178.429,5.755,148.549
C08717=1215.323,113.403,-49.667,-178.431,5.754,148.549
C08718=1215.328,113.154,-49.648,-178.434,5.753,148.550
C08719=1215.332,112.905,-49.629,-178.437,5.752,148.550
C08720=1215.337,112.656,-49.609,-178.439,5.751,148.551
C08721=1215.342,112.406,-49.590,-178.441,5.750,148.551
C08722=1215.346,112.158,-49.571,-178.445,5.749,148.552
C08723=1215.351,111.908,-49.551,-178.447,5.748,148.553
C08724=1215.357,111.659,-49.533,-178.449,5.747,148.553
C08725=1215.361,111.409,-49.514,-178.452,5.745,148.554
C08726=1215.366,111.160,-49.495,-178.455,5.745,148.554
C08727=1215.371,110.911,-49.475,-178.457,5.744,148.555
C08728=1215.376,110.662,-49.456,-178.460,5.742,148.555
C08729=1215.380,110.413,-49.436,-178.463,5.742,148.556
C08730=1215.386,110.164,-49.417,-178.465,5.741,148.556
C08731=1215.390,109.914,-49.399,-178.468,5.739,148.557
C08732=1215.395,109.664,-49.379,-178.470,5.738,148.557
C08733=1215.399,109.416,-49.361,-178.473,5.738,148.558
C08734=1215.404,109.166,-49.341,-178.475,5.736,148.558
C08735=1215.409,108.917,-49.322,-178.478,5.735,148.559
C08736=1215.414,108.668,-49.303,-178.481,5.735,148.560
C08737=1215.419,108.419,-49.284,-178.483,5.733,148.560
C08738=1215.423,108.169,-49.265,-178.486,5.732,148.561
C08739=1215.428,107.921,-49.246,-178.488,5.731,148.561
C08740=1215.434,107.652,-49.226,-178.491,5.730,148.562
C08741=1215.439,107.383,-49.204,-178.494,5.729,148.562
C08742=1215.444,107.116,-49.184,-178.496,5.728,148.563
C08743=1215.449,106.846,-49.164,-178.499,5.727,148.563
C08744=1215.454,106.598,-49.145,-178.502,5.726,148.564
C08745=1215.458,106.348,-49.126,-178.504,5.725,148.564
C08746=1215.464,106.099,-49.107,-178.507,5.724,148.565
C08747=1215.468,105.850,-49.088,-178.510,5.723,148.566
C08748=1215.473,105.601,-49.069,-178.512,5.722,148.566
C08749=1215.478,105.351,-49.050,-178.515,5.721,148.567
C08750=1215.483,105.102,-49.031,-178.517,5.720,148.567
C08751=1215.488,104.853,-49.012,-178.520,5.719,148.568
C08752=1215.493,104.603,-48.993,-178.522,5.718,148.568
C08753=1215.497,104.355,-48.975,-178.525,5.717,148.569
C08754=1215.502,104.105,-48.956,-178.528,5.717,148.570
C08755=1215.507,103.856,-48.937,-178.530,5.715,148.570
C08756=1215.512,103.606,-48.917,-178.533,5.714,148.571
C08757=1215.517,103.357,-48.899,-178.535,5.713,148.571
C08758=1215.521,103.109,-48.881,-178.538,5.712,148.572
C08759=1215.526,102.858,-48.862,-178.541,5.711,148.572
C08760=1215.531,102.610,-48.843,-178.543,5.710,148.573
C08761=1215.536,102.360,-48.824,-178.546,5.710,148.573
C08762=1215.541,102.111,-48.805,-178.548,5.708,148.574
C08763=1215.546,101.862,-48.786,-178.551,5.707,148.574
C08764=1215.550,101.612,-48.768,-178.553,5.707,148.575
C08765=1215.555,101.364,-48.749,-178.556,5.705,148.575
C08766=1215.561,101.114,-48.731,-178.559,5.704,148.576
C08767=1215.565,100.865,-48.712,-178.561,5.703,148.577
C08768=1215.570,100.616,-48.693,-178.564,5.703,148.577
C08769=1215.575,100.366,-48.675,-178.567,5.701,148.578
C08770=1215.579,100.117,-48.656,-178.569,5.700,148.578
C08771=1215.585,99.868,-48.637,-178.571,5.700,148.579
C08772=1215.589,99.618,-48.618,-178.574,5.699,148.579
C08773=1215.594,99.369,-48.600,-178.577,5.698,148.580
C08774=1215.599,99.120,-48.581,-178.579,5.697,148.581
C08775=1215.603,98.871,-48.563,-178.582,5.696,148.581
C08776=1215.608,98.622,-48.544,-178.585,5.695,148.582
C08777=1215.614,98.373,-48.525,-178.587,5.694,148.582
C08778=1215.618,98.123,-48.507,-178.589,5.693,148.583
C08779=1215.622,97.874,-48.488,-178.592,5.692,148.583
C08780=1215.628,97.625,-48.470,-178.595,5.691,148.584
C08781=1215.632,97.375,-48.451,-178.597,5.690,148.584
C08782=1215.637,97.126,-48.433,-178.600,5.689,148.585
C08783=1215.643,96.877,-48.414,-178.602,5.689,148.585
C08784=1215.647,96.627,-48.396,-178.605,5.687,148.586
C08785=1215.652,96.378,-48.377,-178.607,5.686,148.587
C08786=1215.657,96.129,-48.359,-178.610,5.686,148.587
C08787=1215.662,95.880,-48.341,-178.613,5.685,148.588
C08788=1215.666,95.630,-48.322,-178.615,5.683,148.588
C08789=1215.671,95.381,-48.304,-178.618,5.683,148.589
C08790=1215.677,95.132,-48.285,-178.620,5.682,148.589
C08791=1215.681,94.882,-48.266,-178.623,5.681,148.590
C08792=1215.686,94.633,-48.248,-178.626,5.680,148.591
C08793=1215.691,94.384,-48.230,-178.628,5.679,148.591
C08794=1215.696,94.135,-48.212,-178.631,5.678,148.592
C08795=1215.700,93.885,-48.192,-178.633,5.678,148.592
C08796=1215.705,93.636,-48.174,-178.635,5.677,148.593
C08797=1215.710,93.387,-48.156,-178.639,5.675,148.593
C08798=1215.715,93.138,-48.138,-178.641,5.675,148.594
C08799=1215.719,92.888,-48.120,-178.643,5.674,148.594
C08800=1215.725,92.639,-48.101,-178.646,5.673,148.595
C08801=1215.730,92.390,-48.083,-178.649,5.671,148.596
C08802=1215.734,92.141,-48.065,-178.651,5.671,148.596
C08803=1215.739,91.891,-48.046,-178.654,5.670,148.597
C08804=1215.744,91.642,-48.028,-178.656,5.669,148.597
C08805=1215.749,91.392,-48.010,-178.659,5.669,148.598
C08806=1215.754,91.144,-47.991,-178.662,5.667,148.599
C08807=1215.759,90.894,-47.973,-178.664,5.666,148.599
C08808=1215.763,90.645,-47.955,-178.667,5.666,148.600
C08809=1215.768,90.395,-47.937,-178.669,5.665,148.600
C08810=1215.773,90.146,-47.919,-178.672,5.663,148.601
C08811=1215.778,89.897,-47.901,-178.675,5.663,148.601
C08812=1215.783,89.648,-47.883,-178.677,5.662,148.602
C08813=1215.787,89.398,-47.865,-178.679,5.661,148.602
C08814=1215.793,89.148,-47.846,-178.682,5.661,148.603
C08815=1215.798,88.899,-47.828,-178.685,5.659,148.604
C08816=1215.803,88.650,-47.810,-178.687,5.658,148.604
C08817=1215.808,88.401,-47.792,-178.690,5.658,148.605
C08818=1215.812,88.152,-47.773,-178.693,5.657,148.605
C08819=1215.816,87.903,-47.755,-178.695,5.656,148.606
C08820=1215.821,87.653,-47.737,-178.698,5.655,148.606
C08821=1215.826,87.404,-47.719,-178.700,5.654,148.607
C08822=1215.831,87.155,-47.701,-178.703,5.653,148.608
C08823=1215.836,86.906,-47.683,-178.705,5.653,148.608
C08824=1215.841,86.656,-47.666,-178.708,5.652,148.609
C08825=1215.846,86.407,-47.648,-178.711,5.650,148.609
C08826=1215.851,86.157,-47.630,-178.713,5.650,148.610
C08827=1215.855,85.908,-47.612,-178.716,5.649,148.611
C08828=1215.860,85.659,-47.594,-178.718,5.648,148.611
C08829=1215.865,85.409,-47.576,-178.721,5.648,148.612
C08830=1215.870,85.160,-47.558,-178.724,5.646,148.612
C08831=1215.875,84.911,-47.540,-178.726,5.645,148.613
C08832=1215.880,84.662,-47.522,-178.729,5.645,148.613
C08833=1215.885,84.413,-47.504,-178.731,5.644,148.614
C08834=1215.890,84.164,-47.486,-178.733,5.643,148.614
C08835=1215.894,83.914,-47.467,-178.736,5.643,148.615
C08836=1215.899,83.664,-47.450,-178.739,5.641,148.616
C08837=1215.904,83.415,-47.432,-178.741,5.640,148.616
C08838=1215.909,83.166,-47.414,-178.744,5.640,148.617
C08839=1215.914,82.916,-47.396,-178.746,5.639,148.618
C08840=1215.919,82.667,-47.378,-178.749,5.638,148.618
C08841=1215.924,82.418,-47.360,-178.751,5.638,148.619
C08842=1215.929,82.168,-47.343,-178.754,5.636,148.619
C08843=1215.934,81.919,-47.325,-178.757,5.635,148.620
C08844=1215.939,81.651,-47.306,-178.759,5.635,148.620
C08845=1215.944,81.383,-47.286,-178.762,5.634,148.621
C08846=1215.950,81.114,-47.267,-178.765,5.633,148.622
C08847=1215.955,80.845,-47.248,-178.768,5.632,148.622
C08848=1215.960,80.596,-47.230,-178.770,5.632,148.623
C08849=1215.964,80.347,-47.213,-178.772,5.631,148.623
C08850=1215.969,80.098,-47.195,-178.776,5.629,148.624
C08851=1215.974,79.848,-47.177,-178.778,5.629,148.625
C08852=1215.979,79.599,-47.159,-178.781,5.628,148.625
C08853=1215.984,79.349,-47.142,-178.783,5.627,148.626
C08854=1215.989,79.100,-47.124,-178.786,5.627,148.626
C08855=1215.994,78.851,-47.106,-178.788,5.626,148.627
C08856=1215.998,78.602,-47.090,-178.791,5.624,148.627
C08857=1216.003,78.352,-47.072,-178.794,5.624,148.628
C08858=1216.008,78.103,-47.054,-178.796,5.623,148.629
C08859=1216.013,77.853,-47.036,-178.798,5.622,148.629
C08860=1216.018,77.604,-47.018,-178.801,5.622,148.630
C08861=1216.023,77.355,-47.000,-178.804,5.621,148.631
C08862=1216.028,77.106,-46.984,-178.806,5.620,148.631
C08863=1216.033,76.856,-46.966,-178.809,5.619,148.632
C08864=1216.037,76.607,-46.948,-178.812,5.618,148.632
C08865=1216.043,76.357,-46.930,-178.814,5.617,148.633
C08866=1216.047,76.109,-46.913,-178.816,5.617,148.633
C08867=1216.052,75.859,-46.896,-178.819,5.616,148.634
C08868=1216.057,75.610,-46.878,-178.822,5.615,148.635
C08869=1216.062,75.360,-46.860,-178.824,5.615,148.635
C08870=1216.066,75.111,-46.843,-178.827,5.613,148.636
C08871=1216.071,74.862,-46.825,-178.830,5.612,148.636
C08872=1216.077,74.612,-46.808,-178.832,5.612,148.637
C08873=1216.081,74.363,-46.790,-178.834,5.611,148.638
C08874=1216.086,74.113,-46.773,-178.837,5.610,148.638
C08875=1216.091,73.864,-46.755,-178.840,5.610,148.639
C08876=1216.097,73.615,-46.738,-178.842,5.609,148.639
C08877=1216.102,73.366,-46.720,-178.844,5.608,148.640
C08878=1216.106,73.116,-46.704,-178.848,5.607,148.641
C08879=1216.111,72.867,-46.686,-178.850,5.606,148.641
C08880=1216.116,72.617,-46.668,-178.853,5.606,148.642
C08881=1216.120,72.369,-46.651,-178.855,5.605,148.642
C08882=1216.126,72.119,-46.634,-178.858,5.604,148.643
C08883=1216.130,71.870,-46.616,-178.860,5.604,148.644
C08884=1216.135,71.620,-46.599,-178.862,5.603,148.644
C08885=1216.140,71.371,-46.581,-178.865,5.602,148.645
C08886=1216.145,71.121,-46.564,-178.868,5.602,148.645
C08887=1216.150,70.872,-46.548,-178.871,5.600,148.646
C08888=1216.155,70.623,-46.530,-178.873,5.599,148.646
C08889=1216.160,70.373,-46.512,-178.876,5.599,148.647
C08890=1216.164,70.125,-46.495,-178.878,5.598,148.648
C08891=1216.170,69.875,-46.478,-178.881,5.598,148.648
C08892=1216.174,69.625,-46.461,-178.883,5.597,148.649
C08893=1216.179,69.376,-46.443,-178.886,5.596,148.650
C08894=1216.184,69.126,-46.426,-178.888,5.596,148.650
C08895=1216.189,68.877,-46.410,-178.891,5.595,148.651
C08896=1216.194,68.628,-46.392,-178.893,5.594,148.651
C08897=1216.199,68.379,-46.375,-178.896,5.593,148.652
C08898=1216.204,68.129,-46.358,-178.899,5.592,148.653
C08899=1216.208,67.880,-46.340,-178.901,5.592,148.653
C08900=1216.213,67.630,-46.323,-178.904,5.591,148.654
C08901=1216.219,67.381,-46.306,-178.906,5.590,148.654
C08902=1216.224,67.132,-46.289,-178.909,5.589,148.655
C08903=1216.229,66.883,-46.271,-178.911,5.589,148.656
C08904=1216.233,66.633,-46.255,-178.914,5.588,148.656
C08905=1216.238,66.383,-46.237,-178.916,5.587,148.657
C08906=1216.242,66.134,-46.220,-178.919,5.587,148.657
C08907=1216.248,65.885,-46.203,-178.921,5.586,148.658
C08908=1216.253,65.636,-46.187,-178.924,5.585,148.659
C08909=1216.258,65.386,-46.169,-178.927,5.584,148.659
C08910=1216.262,65.137,-46.153,-178.929,5.583,148.660
C08911=1216.267,64.887,-46.135,-178.932,5.583,148.661
C08912=1216.272,64.639,-46.118,-178.934,5.582,148.661
C08913=1216.278,64.389,-46.101,-178.937,5.581,148.662
C08914=1216.282,64.139,-46.084,-178.939,5.581,148.662
C08915=1216.287,63.890,-46.067,-178.942,5.580,148.663
C08916=1216.292,63.641,-46.050,-178.944,5.579,148.663
C08917=1216.297,63.392,-46.033,-178.947,5.579,148.664
C08918=1216.302,63.142,-46.016,-178.950,5.578,148.665
C08919=1216.307,62.892,-45.999,-178.952,5.578,148.665
C08920=1216.312,62.643,-45.982,-178.955,5.577,148.666
C08921=1216.317,62.394,-45.966,-178.958,5.575,148.666
C08922=1216.322,62.144,-45.949,-178.960,5.575,148.667
C08923=1216.326,61.895,-45.932,-178.963,5.574,148.668
C08924=1216.332,61.645,-45.915,-178.965,5.574,148.668
C08925=1216.336,61.397,-45.898,-178.968,5.573,148.669
C08926=1216.342,61.147,-45.880,-178.970,5.572,148.670
C08927=1216.346,60.898,-45.864,-178.973,5.572,148.670
C08928=1216.350,60.648,-45.847,-178.975,5.571,148.671
C08929=1216.356,60.399,-45.830,-178.978,5.570,148.672
C08930=1216.361,60.150,-45.814,-178.980,5.569,148.672
C08931=1216.366,59.900,-45.796,-178.983,5.569,148.673
C08932=1216.371,59.651,-45.780,-178.985,5.568,148.673
C08933=1216.376,59.401,-45.763,-178.988,5.568,148.674
C08934=1216.381,59.152,-45.746,-178.990,5.567,148.674
C08935=1216.385,58.902,-45.729,-178.993,5.566,148.675
C08936=1216.390,58.653,-45.713,-178.996,5.566,148.676
C08937=1216.396,58.404,-45.696,-178.998,5.565,148.676
C08938=1216.400,58.154,-45.679,-179.001,5.565,148.677
C08939=1216.405,57.905,-45.663,-179.004,5.563,148.678
C08940=1216.410,57.656,-45.646,-179.006,5.562,148.678
C08941=1216.415,57.406,-45.629,-179.009,5.562,148.679
C08942=1216.420,57.157,-45.613,-179.011,5.561,148.680
C08943=1216.425,56.907,-45.595,-179.014,5.560,148.680
C08944=1216.430,56.657,-45.579,-179.016,5.560,148.681
C08945=1216.435,56.409,-45.563,-179.019,5.559,148.681
C08946=1216.440,56.159,-45.546,-179.021,5.559,148.682
C08947=1216.445,55.909,-45.529,-179.024,5.558,148.683
C08948=1216.450,55.641,-45.511,-179.027,5.557,148.683
C08949=1216.455,55.373,-45.493,-179.029,5.557,148.684
C08950=1216.461,55.104,-45.476,-179.032,5.556,148.685
C08951=1216.466,54.836,-45.458,-179.035,5.555,148.685
C08952=1216.471,54.587,-45.441,-179.038,5.554,148.686
C08953=1216.476,54.337,-45.424,-179.040,5.554,148.686
C08954=1216.481,54.088,-45.408,-179.043,5.553,148.687
C08955=1216.486,53.838,-45.392,-179.045,5.552,148.688
C08956=1216.490,53.589,-45.375,-179.048,5.552,148.688
C08957=1216.496,53.339,-45.358,-179.051,5.551,148.689
C08958=1216.500,53.090,-45.342,-179.053,5.550,148.690
C08959=1216.506,52.841,-45.326,-179.055,5.550,148.690
C08960=1216.510,52.591,-45.309,-179.058,5.549,148.691
C08961=1216.515,52.342,-45.293,-179.061,5.549,148.692
C08962=1216.521,52.093,-45.276,-179.063,5.548,148.692
C08963=1216.525,51.843,-45.259,-179.065,5.547,148.693
C08964=1216.531,51.594,-45.243,-179.068,5.547,148.693
C08965=1216.535,51.344,-45.227,-179.071,5.546,148.694
C08966=1216.539,51.095,-45.210,-179.073,5.546,148.695
C08967=1216.545,50.845,-45.195,-179.076,5.545,148.695
C08968=1216.550,50.595,-45.177,-179.078,5.544,148.696
C08969=1216.555,50.347,-45.161,-179.081,5.544,148.696
C08970=1216.560,50.097,-45.144,-179.083,5.543,148.697
C08971=1216.565,49.848,-45.129,-179.086,5.542,148.698
C08972=1216.570,49.598,-45.112,-179.089,5.542,148.698
C08973=1216.574,49.349,-45.095,-179.091,5.541,148.699
C08974=1216.579,49.099,-45.080,-179.093,5.540,148.700
C08975=1216.584,48.850,-45.063,-179.096,5.540,148.700
C08976=1216.590,48.601,-45.046,-179.099,5.539,148.701
C08977=1216.594,48.351,-45.030,-179.101,5.539,148.702
C08978=1216.600,48.102,-45.014,-179.104,5.538,148.702
C08979=1216.604,47.852,-44.998,-179.106,5.537,148.703
C08980=1216.609,47.603,-44.982,-179.109,5.537,148.703
C08981=1216.614,47.354,-44.965,-179.111,5.536,148.704
C08982=1216.619,47.104,-44.949,-179.114,5.536,148.705
C08983=1216.624,46.855,-44.933,-179.117,5.535,148.705
C08984=1216.629,46.605,-44.917,-179.119,5.535,148.706
C08985=1216.634,46.356,-44.901,-179.121,5.534,148.706
C08986=1216.639,46.107,-44.884,-179.124,5.533,148.707
C08987=1216.643,45.857,-44.868,-179.127,5.533,148.708
C08988=1216.649,45.608,-44.852,-179.129,5.532,148.708
C08989=1216.653,45.358,-44.836,-179.132,5.531,148.709
C08990=1216.658,45.109,-44.820,-179.134,5.531,148.710
C08991=1216.663,44.859,-44.804,-179.137,5.530,148.710
C08992=1216.668,44.610,-44.787,-179.139,5.529,148.711
C08993=1216.673,44.360,-44.771,-179.142,5.529,148.712
C08994=1216.678,44.112,-44.755,-179.145,5.528,148.712
C08995=1216.683,43.861,-44.739,-179.147,5.528,148.713
C08996=1216.688,43.613,-44.723,-179.149,5.527,148.713
C08997=1216.693,43.363,-44.707,-179.152,5.526,148.714
C08998=1216.698,43.114,-44.691,-179.155,5.526,148.715
C08999=1216.703,42.864,-44.675,-179.157,5.526,148.715
C09000=1216.708,42.614,-44.659,-179.159,5.525,148.716
C09001=1216.713,42.365,-44.642,-179.162,5.525,148.717
C09002=1216.718,42.115,-44.627,-179.164,5.524,148.717
C09003=1216.723,41.867,-44.611,-179.167,5.523,148.718
C09004=1216.728,41.616,-44.595,-179.170,5.523,148.719
C09005=1216.733,41.367,-44.579,-179.172,5.522,148.719
C09006=1216.738,41.118,-44.562,-179.175,5.522,148.720
C09007=1216.743,40.868,-44.547,-179.177,5.521,148.721
C09008=1216.748,40.619,-44.530,-179.180,5.521,148.721
C09009=1216.753,40.369,-44.515,-179.182,5.520,148.722
C09010=1216.758,40.120,-44.499,-179.185,5.519,148.722
C09011=1216.763,39.870,-44.482,-179.188,5.519,148.723
C09012=1216.768,39.621,-44.467,-179.190,5.518,148.724
C09013=1216.772,39.371,-44.451,-179.193,5.518,148.724
C09014=1216.777,39.122,-44.435,-179.195,5.517,148.725
C09015=1216.783,38.873,-44.419,-179.198,5.516,148.725
C09016=1216.787,38.623,-44.403,-179.200,5.516,148.726
C09017=1216.793,38.374,-44.387,-179.203,5.515,148.727
C09018=1216.798,38.125,-44.372,-179.206,5.515,148.728
C09019=1216.803,37.875,-44.356,-179.208,5.514,148.728
C09020=1216.808,37.625,-44.340,-179.211,5.513,148.729
C09021=1216.812,37.376,-44.324,-179.213,5.513,148.730
C09022=1216.817,37.127,-44.308,-179.215,5.513,148.730
C09023=1216.823,36.877,-44.293,-179.218,5.512,148.731
C09024=1216.827,36.627,-44.277,-179.220,5.512,148.731
C09025=1216.833,36.378,-44.261,-179.223,5.511,148.732
C09026=1216.838,36.129,-44.245,-179.226,5.511,148.733
C09027=1216.842,35.879,-44.230,-179.228,5.510,148.733
C09028=1216.847,35.630,-44.214,-179.231,5.510,148.734
C09029=1216.852,35.381,-44.198,-179.233,5.509,148.734
C09030=1216.857,35.131,-44.182,-179.236,5.508,148.735
C09031=1216.863,34.881,-44.166,-179.238,5.508,148.736
C09032=1216.867,34.632,-44.151,-179.241,5.507,148.737
C09033=1216.872,34.382,-44.135,-179.244,5.506,148.737
C09034=1216.877,34.133,-44.120,-179.246,5.506,148.738
C09035=1216.882,33.884,-44.103,-179.249,5.505,148.739
C09036=1216.887,33.634,-44.088,-179.251,5.505,148.739
C09037=1216.892,33.385,-44.072,-179.253,5.505,148.740
C09038=1216.897,33.135,-44.057,-179.256,5.504,148.740
C09039=1216.902,32.885,-44.041,-179.258,5.504,148.741
C09040=1216.907,32.636,-44.026,-179.261,5.503,148.742
C09041=1216.912,32.387,-44.010,-179.264,5.503,148.742
C09042=1216.918,32.137,-43.995,-179.266,5.502,148.743
C09043=1216.922,31.887,-43.979,-179.269,5.502,148.744
C09044=1216.927,31.639,-43.963,-179.271,5.501,148.744
C09045=1216.932,31.390,-43.947,-179.274,5.500,148.745
C09046=1216.937,31.139,-43.931,-179.276,5.500,148.746
C09047=1216.941,30.890,-43.916,-179.279,5.499,148.746
C09048=1216.947,30.641,-43.901,-179.282,5.498,148.747
C09049=1216.952,30.392,-43.885,-179.284,5.498,148.748
C09050=1216.956,30.142,-43.870,-179.286,5.498,148.748
C09051=1216.962,29.892,-43.854,-179.289,5.498,148.749
C09052=1216.967,29.624,-43.837,-179.292,5.497,148.750
C09053=1216.973,29.355,-43.821,-179.294,5.497,148.750
C09054=1216.978,29.087,-43.805,-179.297,5.496,148.751
C09055=1216.983,28.818,-43.788,-179.300,5.495,148.752
C09056=1216.988,28.568,-43.772,-179.302,5.495,148.752
C09057=1216.993,28.318,-43.757,-179.305,5.494,148.753
C09058=1216.999,28.069,-43.742,-179.308,5.494,148.754
C09059=1217.003,27.820,-43.727,-179.310,5.493,148.754
C09060=1217.008,27.570,-43.711,-179.312,5.492,148.755
C09061=1217.013,27.320,-43.695,-179.315,5.492,148.755
C09062=1217.018,27.071,-43.680,-179.318,5.491,148.756
C09063=1217.023,26.822,-43.665,-179.320,5.491,148.757
C09064=1217.028,26.573,-43.650,-179.323,5.490,148.758
C09065=1217.033,26.323,-43.634,-179.326,5.490,148.758
C09066=1217.038,26.073,-43.618,-179.328,5.490,148.759
C09067=1217.043,25.824,-43.603,-179.330,5.490,148.760
C09068=1217.048,25.575,-43.588,-179.332,5.489,148.760
C09069=1217.053,25.325,-43.573,-179.335,5.488,148.761
C09070=1217.058,25.075,-43.557,-179.338,5.488,148.761
C09071=1217.063,24.826,-43.542,-179.340,5.487,148.762
C09072=1217.068,24.576,-43.527,-179.343,5.487,148.763
C09073=1217.073,24.327,-43.511,-179.346,5.486,148.763
C09074=1217.078,24.078,-43.496,-179.348,5.485,148.764
C09075=1217.084,23.828,-43.481,-179.350,5.486,148.765
C09076=1217.088,23.578,-43.466,-179.353,5.485,148.765
C09077=1217.093,23.329,-43.450,-179.355,5.484,148.766
C09078=1217.098,23.080,-43.435,-179.358,5.484,148.767
C09079=1217.103,22.830,-43.420,-179.360,5.483,148.767
C09080=1217.108,22.580,-43.405,-179.363,5.483,148.768
C09081=1217.114,22.331,-43.390,-179.366,5.482,148.769
C09082=1217.118,22.082,-43.375,-179.368,5.482,148.769
C09083=1217.123,21.832,-43.359,-179.370,5.482,148.770
C09084=1217.128,21.582,-43.345,-179.373,5.481,148.771
C09085=1217.133,21.333,-43.329,-179.376,5.481,148.771
C09086=1217.138,21.084,-43.314,-179.378,5.480,148.772
C09087=1217.143,20.834,-43.298,-179.381,5.479,148.772
C09088=1217.148,20.585,-43.284,-179.383,5.479,148.773
C09089=1217.153,20.335,-43.269,-179.386,5.478,148.774
C09090=1217.158,20.086,-43.254,-179.389,5.478,148.775
C09091=1217.163,19.836,-43.239,-179.391,5.478,148.775
C09092=1217.168,19.586,-43.223,-179.393,5.478,148.776
C09093=1217.173,19.337,-43.208,-179.396,5.477,148.777
C09094=1217.179,19.087,-43.194,-179.399,5.477,148.777
C09095=1217.183,18.838,-43.179,-179.401,5.476,148.778
C09096=1217.188,18.589,-43.164,-179.403,5.475,148.778
C09097=1217.194,18.339,-43.149,-179.406,5.475,148.779
C09098=1217.198,18.090,-43.134,-179.408,5.475,148.780
C09099=1217.204,17.840,-43.118,-179.411,5.474,148.780
C09100=1217.208,17.591,-43.104,-179.413,5.474,148.781
C09101=1217.213,17.342,-43.089,-179.416,5.473,148.782
C09102=1217.219,17.092,-43.074,-179.419,5.473,148.782
C09103=1217.223,16.842,-43.059,-179.421,5.472,148.783
C09104=1217.228,16.592,-43.043,-179.424,5.472,148.784
C09105=1217.233,16.343,-43.029,-179.426,5.472,148.785
C09106=1217.238,16.094,-43.014,-179.428,5.471,148.785
C09107=1217.244,15.844,-42.999,-179.431,5.471,148.786
C09108=1217.248,15.594,-42.984,-179.433,5.470,148.786
C09109=1217.253,15.345,-42.970,-179.436,5.470,148.787
C09110=1217.259,15.095,-42.954,-179.439,5.469,148.788
C09111=1217.263,14.846,-42.939,-179.441,5.469,148.788
C09112=1217.268,14.597,-42.925,-179.443,5.469,148.789
C09113=1217.274,14.347,-42.909,-179.446,5.468,148.790
C09114=1217.279,14.097,-42.895,-179.449,5.468,148.790
C09115=1217.283,13.848,-42.880,-179.451,5.467,148.791
C09116=1217.288,13.599,-42.866,-179.454,5.467,148.792
C09117=1217.293,13.349,-42.850,-179.457,5.466,148.792
C09118=1217.298,13.100,-42.836,-179.458,5.466,148.793
C09119=1217.303,12.850,-42.821,-179.461,5.466,148.794
C09120=1217.309,12.600,-42.806,-179.464,5.465,148.794
C09121=1217.314,12.351,-42.792,-179.466,5.465,148.795
C09122=1217.318,12.102,-42.777,-179.469,5.464,148.796
C09123=1217.323,11.852,-42.762,-179.472,5.463,148.796
C09124=1217.329,11.603,-42.747,-179.474,5.464,148.797
C09125=1217.334,11.353,-42.732,-179.476,5.463,148.798
C09126=1217.339,11.103,-42.718,-179.479,5.463,148.798
C09127=1217.343,10.854,-42.703,-179.482,5.462,148.799
C09128=1217.349,10.604,-42.688,-179.484,5.462,148.800
C09129=1217.354,10.355,-42.673,-179.486,5.461,148.800
C09130=1217.359,10.105,-42.659,-179.488,5.461,148.801
C09131=1217.364,9.855,-42.645,-179.491,5.461,148.802
C09132=1217.369,9.606,-42.629,-179.494,5.460,148.802
C09133=1217.374,9.356,-42.615,-179.496,5.460,148.803
C09134=1217.379,9.107,-42.601,-179.499,5.459,148.804
C09135=1217.383,8.858,-42.586,-179.501,5.459,148.804
C09136=1217.389,8.609,-42.572,-179.504,5.459,148.805
C09137=1217.394,8.359,-42.557,-179.506,5.458,148.806
C09138=1217.399,8.109,-42.542,-179.509,5.458,148.806
C09139=1217.404,7.860,-42.528,-179.512,5.457,148.807
